LIN {X 0,Y 145.986,Z 279.775,A -85,B 0,C 180,E1 -25805.523,E2 -25805.523} C_VEL
LIN {X 0,Y 143.96,Z 293.571,A -85,B 0,C 180,E1 -25806.6,E2 -25806.6} C_VEL
LIN {X 0,Y 141.469,Z 306.049,A -85,B 0,C 180,E1 -25808.124,E2 -25808.124} C_VEL
LIN {X 0,Y 138.489,Z 317.193,A -85,B 0,C 180,E1 -25809.967,E2 -25809.967} C_VEL
LIN {X 0,Y 134.632,Z 328.9,A -85,B 0,C 180,E1 -25812.532,E2 -25812.532} C_VEL
LIN {X 0,Y 130.68,Z 339.104,A -85,B 0,C 180,E1 -25815.465,E2 -25815.465} C_VEL
LIN {X 0,Y 126.897,Z 348.015,A -85,B 0,C 180,E1 -25818.822,E2 -25818.822} C_VEL
LIN {X 0,Y 122.512,Z 357.337,A -85,B 0,C 180,E1 -25823.411,E2 -25823.411} C_VEL
LIN {X 0,Y 118.844,Z 364.909,A -85,B 0,C 180,E1 -25828.379,E2 -25828.379} C_VEL
LIN {X 0,Y 115.988,Z 370.741,A -85,B 0,C 180,E1 -25833.473,E2 -25833.473} C_VEL
LIN {X 0,Y 113.868,Z 375.53,A -85,B 0,C 180,E1 -25839.077,E2 -25839.077} C_VEL
LIN {X 0,Y 112.513,Z 378.89,A -85,B 0,C 180,E1 -25844.468,E2 -25844.468} C_VEL
LIN {X 0,Y 111.937,Z 381.142,A -85,B 0,C 180,E1 -25849.658,E2 -25849.658} C_VEL
LIN {X 0,Y 112.099,Z 382.715,A -85,B 0,C 180,E1 -25856.031,E2 -25856.031} C_VEL
LIN {X 0,Y 112.714,Z 383.083,A -85,B 0,C 180,E1 -25859.921,E2 -25859.921} C_VEL
LIN {X 0,Y 113.719,Z 382.989,A -85,B 0,C 180,E1 -25863.794,E2 -25863.794} C_VEL
LIN {X 0,Y 115.187,Z 382.397,A -85,B 0,C 180,E1 -25867.599,E2 -25867.599} C_VEL
LIN {X 0,Y 117.047,Z 381.361,A -85,B 0,C 180,E1 -25871.336,E2 -25871.336} C_VEL
LIN {X 0,Y 120.63,Z 378.856,A -85,B 0,C 180,E1 -25876.738,E2 -25876.738} C_VEL
LIN {X 0,Y 125.188,Z 375.1,A -85,B 0,C 180,E1 -25881.867,E2 -25881.867} C_VEL
LIN {X 0,Y 130.446,Z 370.145,A -85,B 0,C 180,E1 -25886.5,E2 -25886.5} C_VEL
LIN {X 0,Y 136.756,Z 363.485,A -85,B 0,C 180,E1 -25890.884,E2 -25890.884} C_VEL
LIN {X 0,Y 142.45,Z 356.634,A -85,B 0,C 180,E1 -25894.209,E2 -25894.209} C_VEL
LIN {X 0,Y 148.493,Z 348.43,A -85,B 0,C 180,E1 -25897.193,E2 -25897.193} C_VEL
LIN {X 0,Y 154.45,Z 338.924,A -85,B 0,C 180,E1 -25899.801,E2 -25899.801} C_VEL
LIN {X 0,Y 160.006,Z 328.535,A -85,B 0,C 180,E1 -25901.931,E2 -25901.931} C_VEL
LIN {X 0,Y 164.808,Z 317.654,A -85,B 0,C 180,E1 -25903.633,E2 -25903.633} C_VEL
LIN {X 0,Y 168.622,Z 306.885,A -85,B 0,C 180,E1 -25904.913,E2 -25904.913} C_VEL
LIN {X 0,Y 172.048,Z 293.907,A -85,B 0,C 180,E1 -25906.049,E2 -25906.049} C_VEL
LIN {X 0,Y 174.424,Z 281.013,A -85,B 0,C 180,E1 -25906.778,E2 -25906.778} C_VEL
LIN {X 0,Y 176.77,Z 258.578,A -85,B 0,C 180,E1 -25907.541,E2 -25907.541} C_VEL
LIN {X 0,Y 173.643,Z 251.901,A -85,B 0,C 180,E1 -25910.486,E2 -25910.486} C_VEL
LIN {X 0,Y 171.117,Z 247.12,A -85,B 0,C 180,E1 -25913.202,E2 -25913.202} C_VEL
LIN {X 0,Y 169.506,Z 244.096,A -85,B 0,C 180,E1 -25915.245,E2 -25915.245} C_VEL
LIN {X 0,Y 168.036,Z 241.322,A -85,B 0,C 180,E1 -25917.404,E2 -25917.404} C_VEL
LIN {X 0,Y 165.952,Z 237.408,A -85,B 0,C 180,E1 -25921.359,E2 -25921.359} C_VEL
LIN {X 0,Y 164.008,Z 233.239,A -85,B 0,C 180,E1 -25929.872,E2 -25929.872} C_VEL
LIN {X 0,Y 163.962,Z 233.673,A -85,B 0,C 180,E1 -25931.717,E2 -25931.717} C_VEL
LIN {X 0,Y 165.845,Z 237.96,A -85,B 0,C 180,E1 -25940.094,E2 -25940.094} C_VEL
LIN {X 0,Y 166.766,Z 239.887,A -85,B 0,C 180,E1 -25942.101,E2 -25942.101} C_VEL
LIN {X 0,Y 168.245,Z 242.318,A -85,B 0,C 180,E1 -25944.531,E2 -25944.531} C_VEL
LIN {X 0,Y 170.324,Z 247.29,A -85,B 0,C 180,E1 -25947.577,E2 -25947.577} C_VEL
LIN {X 0,Y 172.572,Z 252.652,A -85,B 0,C 180,E1 -25950.247,E2 -25950.247} C_VEL
LIN {X 0,Y 175.387,Z 260.766,A -85,B 0,C 180,E1 -25953.254,E2 -25953.254} C_VEL
LIN {X 0,Y 176.349,Z 263.654,A -85,B 0,C 180,E1 -25954.176,E2 -25954.176} C_VEL
LIN {X 0,Y 173.818,Z 287.836,A -85,B 0,C 180,E1 -25955.046,E2 -25955.046} C_VEL
LIN {X 0,Y 171.228,Z 301.026,A -85,B 0,C 180,E1 -25955.774,E2 -25955.774} C_VEL
LIN {X 0,Y 167.566,Z 313.569,A -85,B 0,C 180,E1 -25956.757,E2 -25956.757} C_VEL
LIN {X 0,Y 162.982,Z 325.554,A -85,B 0,C 180,E1 -25958.098,E2 -25958.098} C_VEL
LIN {X 0,Y 157.717,Z 336.638,A -85,B 0,C 180,E1 -25959.766,E2 -25959.766} C_VEL
LIN {X 0,Y 152.225,Z 346.648,A -85,B 0,C 180,E1 -25961.887,E2 -25961.887} C_VEL
LIN {X 0,Y 145.678,Z 356.545,A -85,B 0,C 180,E1 -25964.636,E2 -25964.636} C_VEL
LIN {X 0,Y 138.987,Z 365.314,A -85,B 0,C 180,E1 -25967.934,E2 -25967.934} C_VEL
LIN {X 0,Y 132.924,Z 372.398,A -85,B 0,C 180,E1 -25971.593,E2 -25971.593} C_VEL
LIN {X 0,Y 126.85,Z 378.898,A -85,B 0,C 180,E1 -25976.356,E2 -25976.356} C_VEL
LIN {X 0,Y 122.22,Z 383.244,A -85,B 0,C 180,E1 -25980.741,E2 -25980.741} C_VEL
LIN {X 0,Y 118.416,Z 386.557,A -85,B 0,C 180,E1 -25985.453,E2 -25985.453} C_VEL
LIN {X 0,Y 114.696,Z 389.513,A -85,B 0,C 180,E1 -25992.16,E2 -25992.16} C_VEL
LIN {X 0,Y 113.54,Z 390.406,A -85,B 0,C 180,E1 -25995.665,E2 -25995.665} C_VEL
LIN {X 0,Y 112.267,Z 390.977,A -85,B 0,C 180,E1 -26002.808,E2 -26002.808} C_VEL
LIN {X 0,Y 112.199,Z 390.696,A -85,B 0,C 180,E1 -26006.409,E2 -26006.409} C_VEL
LIN {X 0,Y 112.393,Z 390.029,A -85,B 0,C 180,E1 -26010.001,E2 -26010.001} C_VEL
LIN {X 0,Y 112.211,Z 388.885,A -85,B 0,C 180,E1 -26013.592,E2 -26013.592} C_VEL
LIN {X 0,Y 112.526,Z 386.385,A -85,B 0,C 180,E1 -26018.984,E2 -26018.984} C_VEL
LIN {X 0,Y 113.513,Z 382.837,A -85,B 0,C 180,E1 -26024.34,E2 -26024.34} C_VEL
LIN {X 0,Y 115.322,Z 378.149,A -85,B 0,C 180,E1 -26029.585,E2 -26029.585} C_VEL
LIN {X 0,Y 118.066,Z 372.192,A -85,B 0,C 180,E1 -26034.626,E2 -26034.626} C_VEL
LIN {X 0,Y 121.163,Z 365.534,A -85,B 0,C 180,E1 -26038.983,E2 -26038.983} C_VEL
LIN {X 0,Y 125.108,Z 357.123,A -85,B 0,C 180,E1 -26043.211,E2 -26043.211} C_VEL
LIN {X 0,Y 129.16,Z 347.899,A -85,B 0,C 180,E1 -26046.767,E2 -26046.767} C_VEL
LIN {X 0,Y 130.848,Z 343.784,A -85,B 0,C 180,E1 -26048.07,E2 -26048.07} C_VEL
LIN {X 0,Y 132.173,Z 339.134,A -85,B 0,C 180,E1 -26049.556,E2 -26049.556} C_VEL
LIN {X 0,Y 132.686,Z 331.21,A -85,B 0,C 180,E1 -26052.14,E2 -26052.14} C_VEL
LIN {X 0,Y 133.11,Z 322.867,A -85,B 0,C 180,E1 -26054.455,E2 -26054.455} C_VEL
LIN {X 0,Y 134.225,Z 317.564,A -85,B 0,C 180,E1 -26055.467,E2 -26055.467} C_VEL
LIN {X 0,Y 137.116,Z 306.394,A -85,B 0,C 180,E1 -26056.921,E2 -26056.921} C_VEL
LIN {X 0,Y 139.525,Z 293.458,A -85,B 0,C 180,E1 -26058.121,E2 -26058.121} C_VEL
LIN {X 0,Y 140.978,Z 280.384,A -85,B 0,C 180,E1 -26058.888,E2 -26058.888} C_VEL
LIN {X 0,Y 143.348,Z 248.743,A -85,B 0,C 180,E1 -26060.277,E2 -26060.277} C_VEL
LIN {X 0,Y 140.143,Z 238.589,A -85,B 0,C 180,E1 -26062.259,E2 -26062.259} C_VEL
LIN {X 0,Y 135.355,Z 226.534,A -85,B 0,C 180,E1 -26065.28,E2 -26065.28} C_VEL
LIN {X 0,Y 131.392,Z 217.778,A -85,B 0,C 180,E1 -26067.979,E2 -26067.979} C_VEL
LIN {X 0,Y 125.669,Z 208.745,A -85,B 0,C 180,E1 -26072.069,E2 -26072.069} C_VEL
LIN {X 0,Y 122.802,Z 204.727,A -85,B 0,C 180,E1 -26074.378,E2 -26074.378} C_VEL
LIN {X 0,Y 120.101,Z 200.884,A -85,B 0,C 180,E1 -26076.755,E2 -26076.755} C_VEL
LIN {X 0,Y 117.536,Z 197.763,A -85,B 0,C 180,E1 -26079.202,E2 -26079.202} C_VEL
LIN {X 0,Y 116.453,Z 196.028,A -85,B 0,C 180,E1 -26080.382,E2 -26080.382} C_VEL
LIN {X 0,Y 113.988,Z 193.648,A -85,B 0,C 180,E1 -26083.083,E2 -26083.083} C_VEL
LIN {X 0,Y 112.537,Z 190.796,A -85,B 0,C 180,E1 -26085.069,E2 -26085.069} C_VEL
LIN {X 0,Y 109.957,Z 188.848,A -85,B 0,C 180,E1 -26088.575,E2 -26088.575} C_VEL
LIN {X 0,Y 108.543,Z 186.343,A -85,B 0,C 180,E1 -26091.151,E2 -26091.151} C_VEL
LIN {X 0,Y 108.268,Z 184.955,A -85,B 0,C 180,E1 -26092.068,E2 -26092.068} C_VEL
LIN {X 0,Y 108.9,Z 184.896,A -85,B 0,C 180,E1 -26099.997,E2 -26099.997} C_VEL
LIN {X 0,Y 108.292,Z 184.978,A -85,B 0,C 180,E1 -26107.455,E2 -26107.455} C_VEL
LIN {X 0,Y 108.139,Z 184.981,A -85,B 0,C 180,E1 -26112.87,E2 -26112.87} C_VEL
LIN {X 0,Y 107.859,Z 185.022,A -85,B 0,C 180,E1 -26119.01,E2 -26119.01} C_VEL
LIN {X 0,Y 107.801,Z 185.034,A -85,B 0,C 180,E1 -26124.114,E2 -26124.114} C_VEL
LIN {X 0,Y 107.787,Z 185.047,A -85,B 0,C 180,E1 -26129.944,E2 -26129.944} C_VEL
LIN {X 0,Y 108.51,Z 187.423,A -85,B 0,C 180,E1 -26131.647,E2 -26131.647} C_VEL
LIN {X 0,Y 110.636,Z 189.968,A -85,B 0,C 180,E1 -26135.129,E2 -26135.129} C_VEL
LIN {X 0,Y 112.558,Z 191.06,A -85,B 0,C 180,E1 -26137.607,E2 -26137.607} C_VEL
LIN {X 0,Y 114.12,Z 193.989,A -85,B 0,C 180,E1 -26139.708,E2 -26139.708} C_VEL
LIN {X 0,Y 116.764,Z 196.565,A -85,B 0,C 180,E1 -26142.579,E2 -26142.579} C_VEL
LIN {X 0,Y 119.043,Z 200.028,A -85,B 0,C 180,E1 -26144.939,E2 -26144.939} C_VEL
LIN {X 0,Y 120.634,Z 201.729,A -85,B 0,C 180,E1 -26146.364,E2 -26146.364} C_VEL
LIN {X 0,Y 124.148,Z 206.696,A -85,B 0,C 180,E1 -26149.35,E2 -26149.35} C_VEL
LIN {X 0,Y 128.72,Z 213.396,A -85,B 0,C 180,E1 -26152.8,E2 -26152.8} C_VEL
LIN {X 0,Y 134.828,Z 223.62,A -85,B 0,C 180,E1 -26156.836,E2 -26156.836} C_VEL
LIN {X 0,Y 140.731,Z 234.972,A -85,B 0,C 180,E1 -26160.317,E2 -26160.317} C_VEL
LIN {X 0,Y 143.827,Z 241.661,A -85,B 0,C 180,E1 -26162.006,E2 -26162.006} C_VEL
LIN {X 0,Y 140.706,Z 279.337,A -85,B 0,C 180,E1 -26163.637,E2 -26163.637} C_VEL
LIN {X 0,Y 138.696,Z 292.716,A -85,B 0,C 180,E1 -26164.663,E2 -26164.663} C_VEL
LIN {X 0,Y 136.078,Z 305.504,A -85,B 0,C 180,E1 -26166.203,E2 -26166.203} C_VEL
LIN {X 0,Y 132.691,Z 317.65,A -85,B 0,C 180,E1 -26168.237,E2 -26168.237} C_VEL
LIN {X 0,Y 128.676,Z 329.311,A -85,B 0,C 180,E1 -26170.87,E2 -26170.87} C_VEL
LIN {X 0,Y 124.819,Z 338.762,A -85,B 0,C 180,E1 -26173.648,E2 -26173.648} C_VEL
LIN {X 0,Y 120.554,Z 348.369,A -85,B 0,C 180,E1 -26177.371,E2 -26177.371} C_VEL
LIN {X 0,Y 115.939,Z 357.673,A -85,B 0,C 180,E1 -26182.16,E2 -26182.16} C_VEL
LIN {X 0,Y 112.656,Z 364.034,A -85,B 0,C 180,E1 -26186.463,E2 -26186.463} C_VEL
LIN {X 0,Y 109.483,Z 370.163,A -85,B 0,C 180,E1 -26191.839,E2 -26191.839} C_VEL
LIN {X 0,Y 107.176,Z 375.01,A -85,B 0,C 180,E1 -26197.535,E2 -26197.535} C_VEL
LIN {X 0,Y 105.595,Z 378.69,A -85,B 0,C 180,E1 -26203.47,E2 -26203.47} C_VEL
LIN {X 0,Y 104.822,Z 381.467,A -85,B 0,C 180,E1 -26210.183,E2 -26210.183} C_VEL
LIN {X 0,Y 105.241,Z 383.128,A -85,B 0,C 180,E1 -26217.869,E2 -26217.869} C_VEL
LIN {X 0,Y 106.041,Z 383.377,A -85,B 0,C 180,E1 -26222.019,E2 -26222.019} C_VEL
LIN {X 0,Y 108.552,Z 382.675,A -85,B 0,C 180,E1 -26229.026,E2 -26229.026} C_VEL
LIN {X 0,Y 111.246,Z 381.268,A -85,B 0,C 180,E1 -26234.021,E2 -26234.021} C_VEL
LIN {X 0,Y 115.363,Z 378.544,A -85,B 0,C 180,E1 -26239.597,E2 -26239.597} C_VEL
LIN {X 0,Y 120.416,Z 374.603,A -85,B 0,C 180,E1 -26244.795,E2 -26244.795} C_VEL
LIN {X 0,Y 125.771,Z 369.863,A -85,B 0,C 180,E1 -26249.14,E2 -26249.14} C_VEL
LIN {X 0,Y 131.948,Z 363.75,A -85,B 0,C 180,E1 -26253.145,E2 -26253.145} C_VEL
LIN {X 0,Y 137.968,Z 356.91,A -85,B 0,C 180,E1 -26256.478,E2 -26256.478} C_VEL
LIN {X 0,Y 144.054,Z 349.03,A -85,B 0,C 180,E1 -26259.361,E2 -26259.361} C_VEL
LIN {X 0,Y 150.534,Z 339.207,A -85,B 0,C 180,E1 -26262.035,E2 -26262.035} C_VEL
LIN {X 0,Y 156.561,Z 328.354,A -85,B 0,C 180,E1 -26264.211,E2 -26264.211} C_VEL
LIN {X 0,Y 161.296,Z 317.944,A -85,B 0,C 180,E1 -26265.807,E2 -26265.807} C_VEL
LIN {X 0,Y 165.379,Z 306.809,A -85,B 0,C 180,E1 -26267.098,E2 -26267.098} C_VEL
LIN {X 0,Y 168.937,Z 293.767,A -85,B 0,C 180,E1 -26268.201,E2 -26268.201} C_VEL
LIN {X 0,Y 171.318,Z 281.228,A -85,B 0,C 180,E1 -26268.889,E2 -26268.889} C_VEL
LIN {X 0,Y 173.408,Z 262.063,A -85,B 0,C 180,E1 -26269.548,E2 -26269.548} C_VEL
LIN {X 0,Y 170.005,Z 254.678,A -85,B 0,C 180,E1 -26273.251,E2 -26273.251} C_VEL
LIN {X 0,Y 167.444,Z 249.727,A -85,B 0,C 180,E1 -26276.718,E2 -26276.718} C_VEL
LIN {X 0,Y 166.375,Z 247.659,A -85,B 0,C 180,E1 -26278.454,E2 -26278.454} C_VEL
LIN {X 0,Y 164.656,Z 244.108,A -85,B 0,C 180,E1 -26282.134,E2 -26282.134} C_VEL
LIN {X 0,Y 163.074,Z 240.291,A -85,B 0,C 180,E1 -26289.929,E2 -26289.929} C_VEL
LIN {X 0,Y 163.029,Z 241.202,A -85,B 0,C 180,E1 -26292.449,E2 -26292.449} C_VEL
LIN {X 0,Y 164.921,Z 245.281,A -85,B 0,C 180,E1 -26300.2,E2 -26300.2} C_VEL
LIN {X 0,Y 166.736,Z 248.974,A -85,B 0,C 180,E1 -26303.769,E2 -26303.769} C_VEL
LIN {X 0,Y 168.544,Z 253.593,A -85,B 0,C 180,E1 -26306.645,E2 -26306.645} C_VEL
LIN {X 0,Y 170.618,Z 259.175,A -85,B 0,C 180,E1 -26309.371,E2 -26309.371} C_VEL
LIN {X 0,Y 173.009,Z 266.682,A -85,B 0,C 180,E1 -26312.165,E2 -26312.165} C_VEL
LIN {X 0,Y 170.736,Z 287.3,A -85,B 0,C 180,E1 -26312.901,E2 -26312.901} C_VEL
LIN {X 0,Y 167.957,Z 301.038,A -85,B 0,C 180,E1 -26313.648,E2 -26313.648} C_VEL
LIN {X 0,Y 164.141,Z 313.583,A -85,B 0,C 180,E1 -26314.604,E2 -26314.604} C_VEL
LIN {X 0,Y 159.437,Z 325.465,A -85,B 0,C 180,E1 -26315.907,E2 -26315.907} C_VEL
LIN {X 0,Y 153.989,Z 336.517,A -85,B 0,C 180,E1 -26317.535,E2 -26317.535} C_VEL
LIN {X 0,Y 148.251,Z 346.498,A -85,B 0,C 180,E1 -26319.615,E2 -26319.615} C_VEL
LIN {X 0,Y 141.99,Z 355.572,A -85,B 0,C 180,E1 -26322.06,E2 -26322.06} C_VEL
LIN {X 0,Y 134.953,Z 364.447,A -85,B 0,C 180,E1 -26325.329,E2 -26325.329} C_VEL
LIN {X 0,Y 128.454,Z 371.634,A -85,B 0,C 180,E1 -26328.964,E2 -26328.964} C_VEL
LIN {X 0,Y 122.72,Z 377.421,A -85,B 0,C 180,E1 -26333.038,E2 -26333.038} C_VEL
LIN {X 0,Y 117.679,Z 382.027,A -85,B 0,C 180,E1 -26337.487,E2 -26337.487} C_VEL
LIN {X 0,Y 113.258,Z 385.576,A -85,B 0,C 180,E1 -26342.265,E2 -26342.265} C_VEL
LIN {X 0,Y 109.708,Z 388.155,A -85,B 0,C 180,E1 -26347.396,E2 -26347.396} C_VEL
LIN {X 0,Y 107.918,Z 389.392,A -85,B 0,C 180,E1 -26350.998,E2 -26350.998} C_VEL
LIN {X 0,Y 105.755,Z 390.64,A -85,B 0,C 180,E1 -26358.501,E2 -26358.501} C_VEL
LIN {X 0,Y 105.107,Z 390.377,A -85,B 0,C 180,E1 -26366.167,E2 -26366.167} C_VEL
LIN {X 0,Y 105.307,Z 389.652,A -85,B 0,C 180,E1 -26370.001,E2 -26370.001} C_VEL
LIN {X 0,Y 105.119,Z 388.453,A -85,B 0,C 180,E1 -26373.834,E2 -26373.834} C_VEL
LIN {X 0,Y 105.509,Z 385.873,A -85,B 0,C 180,E1 -26379.587,E2 -26379.587} C_VEL
LIN {X 0,Y 106.594,Z 382.236,A -85,B 0,C 180,E1 -26385.292,E2 -26385.292} C_VEL
LIN {X 0,Y 108.642,Z 377.46,A -85,B 0,C 180,E1 -26390.843,E2 -26390.843} C_VEL
LIN {X 0,Y 111.585,Z 371.396,A -85,B 0,C 180,E1 -26396.161,E2 -26396.161} C_VEL
LIN {X 0,Y 114.585,Z 365.353,A -85,B 0,C 180,E1 -26400.279,E2 -26400.279} C_VEL
LIN {X 0,Y 119.175,Z 356.083,A -85,B 0,C 180,E1 -26405.099,E2 -26405.099} C_VEL
LIN {X 0,Y 123.518,Z 346.651,A -85,B 0,C 180,E1 -26408.748,E2 -26408.748} C_VEL
LIN {X 0,Y 127.913,Z 336.182,A -85,B 0,C 180,E1 -26411.775,E2 -26411.775} C_VEL
LIN {X 0,Y 132.068,Z 324.552,A -85,B 0,C 180,E1 -26414.304,E2 -26414.304} C_VEL
LIN {X 0,Y 134.225,Z 317.564,A -85,B 0,C 180,E1 -26415.467,E2 -26415.467} C_VEL
LIN {X 0,Y 134.75,Z 313.661,A -85,B 0,C 180,E1 -26416.23,E2 -26416.23} C_VEL
LIN {X 0,Y 133.048,Z 302.423,A -85,B 0,C 180,E1 -26419.114,E2 -26419.114} C_VEL
LIN {X 0,Y 133.322,Z 298.652,A -85,B 0,C 180,E1 -26419.647,E2 -26419.647} C_VEL
LIN {X 0,Y 135.151,Z 286.464,A -85,B 0,C 180,E1 -26420.558,E2 -26420.558} C_VEL
LIN {X 0,Y 138.1,Z 250.25,A -85,B 0,C 180,E1 -26422.206,E2 -26422.206} C_VEL
LIN {X 0,Y 134.343,Z 238.888,A -85,B 0,C 180,E1 -26424.731,E2 -26424.731} C_VEL
LIN {X 0,Y 129.273,Z 226.193,A -85,B 0,C 180,E1 -26428.331,E2 -26428.331} C_VEL
LIN {X 0,Y 126.996,Z 221.599,A -85,B 0,C 180,E1 -26430.011,E2 -26430.011} C_VEL
LIN {X 0,Y 121.975,Z 213.498,A -85,B 0,C 180,E1 -26433.988,E2 -26433.988} C_VEL
LIN {X 0,Y 117.493,Z 206.959,A -85,B 0,C 180,E1 -26438.067,E2 -26438.067} C_VEL
LIN {X 0,Y 114.879,Z 203.515,A -85,B 0,C 180,E1 -26440.799,E2 -26440.799} C_VEL
LIN {X 0,Y 114.009,Z 202.24,A -85,B 0,C 180,E1 -26441.813,E2 -26441.813} C_VEL
LIN {X 0,Y 111.546,Z 199.443,A -85,B 0,C 180,E1 -26444.787,E2 -26444.787} C_VEL
LIN {X 0,Y 110.439,Z 197.355,A -85,B 0,C 180,E1 -26446.417,E2 -26446.417} C_VEL
LIN {X 0,Y 107.981,Z 195.031,A -85,B 0,C 180,E1 -26450.16,E2 -26450.16} C_VEL
LIN {X 0,Y 106.553,Z 192.054,A -85,B 0,C 180,E1 -26453.132,E2 -26453.132} C_VEL
LIN {X 0,Y 103.837,Z 189.952,A -85,B 0,C 180,E1 -26459.754,E2 -26459.754} C_VEL
LIN {X 0,Y 102.207,Z 188.654,A -85,B 0,C 180,E1 -26467.901,E2 -26467.901} C_VEL
LIN {X 0,Y 102.101,Z 188.838,A -85,B 0,C 180,E1 -26473.645,E2 -26473.645} C_VEL
LIN {X 0,Y 106.16,Z 192.173,A -85,B 0,C 180,E1 -26488.814,E2 -26488.814} C_VEL
LIN {X 0,Y 107.533,Z 195.102,A -85,B 0,C 180,E1 -26491.774,E2 -26491.774} C_VEL
LIN {X 0,Y 109.991,Z 197.293,A -85,B 0,C 180,E1 -26495.632,E2 -26495.632} C_VEL
LIN {X 0,Y 110.598,Z 197.854,A -85,B 0,C 180,E1 -26496.474,E2 -26496.474} C_VEL
LIN {X 0,Y 112.763,Z 201.229,A -85,B 0,C 180,E1 -26499.412,E2 -26499.412} C_VEL
LIN {X 0,Y 114.487,Z 202.991,A -85,B 0,C 180,E1 -26501.362,E2 -26501.362} C_VEL
LIN {X 0,Y 117.016,Z 206.654,A -85,B 0,C 180,E1 -26504.112,E2 -26504.112} C_VEL
LIN {X 0,Y 118.159,Z 208.076,A -85,B 0,C 180,E1 -26505.219,E2 -26505.219} C_VEL
LIN {X 0,Y 121.285,Z 212.635,A -85,B 0,C 180,E1 -26508.061,E2 -26508.061} C_VEL
LIN {X 0,Y 125.47,Z 218.96,A -85,B 0,C 180,E1 -26511.442,E2 -26511.442} C_VEL
LIN {X 0,Y 131.311,Z 229.167,A -85,B 0,C 180,E1 -26515.596,E2 -26515.596} C_VEL
LIN {X 0,Y 136.18,Z 238.872,A -85,B 0,C 180,E1 -26518.7,E2 -26518.7} C_VEL
LIN {X 0,Y 138.506,Z 243.986,A -85,B 0,C 180,E1 -26520.091,E2 -26520.091} C_VEL
LIN {X 0,Y 135.339,Z 280.315,A -85,B 0,C 180,E1 -26521.706,E2 -26521.706} C_VEL
LIN {X 0,Y 133.168,Z 294.058,A -85,B 0,C 180,E1 -26522.816,E2 -26522.816} C_VEL
LIN {X 0,Y 130.288,Z 306.924,A -85,B 0,C 180,E1 -26524.434,E2 -26524.434} C_VEL
LIN {X 0,Y 126.493,Z 319.61,A -85,B 0,C 180,E1 -26526.679,E2 -26526.679} C_VEL
LIN {X 0,Y 122.312,Z 330.947,A -85,B 0,C 180,E1 -26529.393,E2 -26529.393} C_VEL
LIN {X 0,Y 117.7,Z 341.534,A -85,B 0,C 180,E1 -26532.809,E2 -26532.809} C_VEL
LIN {X 0,Y 113.405,Z 350.362,A -85,B 0,C 180,E1 -26536.561,E2 -26536.561} C_VEL
LIN {X 0,Y 109.416,Z 357.967,A -85,B 0,C 180,E1 -26540.759,E2 -26540.759} C_VEL
LIN {X 0,Y 105.338,Z 365.423,A -85,B 0,C 180,E1 -26546.174,E2 -26546.174} C_VEL
LIN {X 0,Y 102.086,Z 371.331,A -85,B 0,C 180,E1 -26551.972,E2 -26551.972} C_VEL
LIN {X 0,Y 99.561,Z 376.411,A -85,B 0,C 180,E1 -26558.811,E2 -26558.811} C_VEL
LIN {X 0,Y 98.674,Z 378.418,A -85,B 0,C 180,E1 -26562.337,E2 -26562.337} C_VEL
LIN {X 0,Y 97.969,Z 380.397,A -85,B 0,C 180,E1 -26566.675,E2 -26566.675} C_VEL
LIN {X 0,Y 97.692,Z 381.873,A -85,B 0,C 180,E1 -26571.081,E2 -26571.081} C_VEL
LIN {X 0,Y 97.844,Z 382.922,A -85,B 0,C 180,E1 -26575.529,E2 -26575.529} C_VEL
LIN {X 0,Y 98.765,Z 383.579,A -85,B 0,C 180,E1 -26581.368,E2 -26581.368} C_VEL
LIN {X 0,Y 101.132,Z 383.279,A -85,B 0,C 180,E1 -26588.714,E2 -26588.714} C_VEL
LIN {X 0,Y 103.189,Z 382.459,A -85,B 0,C 180,E1 -26592.927,E2 -26592.927} C_VEL
LIN {X 0,Y 107.3,Z 380.24,A -85,B 0,C 180,E1 -26599.086,E2 -26599.086} C_VEL
LIN {X 0,Y 112.186,Z 376.997,A -85,B 0,C 180,E1 -26604.527,E2 -26604.527} C_VEL
LIN {X 0,Y 118.12,Z 372.407,A -85,B 0,C 180,E1 -26609.624,E2 -26609.624} C_VEL
LIN {X 0,Y 124.911,Z 366.402,A -85,B 0,C 180,E1 -26614.187,E2 -26614.187} C_VEL
LIN {X 0,Y 132.107,Z 358.967,A -85,B 0,C 180,E1 -26618.14,E2 -26618.14} C_VEL
LIN {X 0,Y 139.091,Z 350.599,A -85,B 0,C 180,E1 -26621.333,E2 -26621.333} C_VEL
LIN {X 0,Y 146.136,Z 340.69,A -85,B 0,C 180,E1 -26624.12,E2 -26624.12} C_VEL
LIN {X 0,Y 152.654,Z 329.59,A -85,B 0,C 180,E1 -26626.369,E2 -26626.369} C_VEL
LIN {X 0,Y 158.03,Z 318.383,A -85,B 0,C 180,E1 -26628.067,E2 -26628.067} C_VEL
LIN {X 0,Y 162.263,Z 307.347,A -85,B 0,C 180,E1 -26629.311,E2 -26629.311} C_VEL
LIN {X 0,Y 165.934,Z 294.444,A -85,B 0,C 180,E1 -26630.383,E2 -26630.383} C_VEL
LIN {X 0,Y 168.464,Z 281.635,A -85,B 0,C 180,E1 -26631.073,E2 -26631.073} C_VEL
LIN {X 0,Y 170.269,Z 265.817,A -85,B 0,C 180,E1 -26631.627,E2 -26631.627} C_VEL
LIN {X 0,Y 167.851,Z 260.355,A -85,B 0,C 180,E1 -26634.614,E2 -26634.614} C_VEL
LIN {X 0,Y 165.304,Z 254.823,A -85,B 0,C 180,E1 -26638.591,E2 -26638.591} C_VEL
LIN {X 0,Y 163.471,Z 250.965,A -85,B 0,C 180,E1 -26642.7,E2 -26642.7} C_VEL
LIN {X 0,Y 162.142,Z 247.336,A -85,B 0,C 180,E1 -26649.986,E2 -26649.986} C_VEL
LIN {X 0,Y 162.174,Z 249.055,A -85,B 0,C 180,E1 -26653.808,E2 -26653.808} C_VEL
LIN {X 0,Y 163.712,Z 252.146,A -85,B 0,C 180,E1 -26659.638,E2 -26659.638} C_VEL
LIN {X 0,Y 165.203,Z 255.442,A -85,B 0,C 180,E1 -26662.885,E2 -26662.885} C_VEL
LIN {X 0,Y 166.911,Z 260.166,A -85,B 0,C 180,E1 -26665.843,E2 -26665.843} C_VEL
LIN {X 0,Y 169.071,Z 266.801,A -85,B 0,C 180,E1 -26668.952,E2 -26668.952} C_VEL
LIN {X 0,Y 169.939,Z 269.913,A -85,B 0,C 180,E1 -26670.091,E2 -26670.091} C_VEL
LIN {X 0,Y 167.742,Z 288.204,A -85,B 0,C 180,E1 -26670.739,E2 -26670.739} C_VEL
LIN {X 0,Y 165.238,Z 300.051,A -85,B 0,C 180,E1 -26671.362,E2 -26671.362} C_VEL
LIN {X 0,Y 161.798,Z 311.475,A -85,B 0,C 180,E1 -26672.176,E2 -26672.176} C_VEL
LIN {X 0,Y 157.555,Z 322.353,A -85,B 0,C 180,E1 -26673.241,E2 -26673.241} C_VEL
LIN {X 0,Y 151.898,Z 333.904,A -85,B 0,C 180,E1 -26674.79,E2 -26674.79} C_VEL
LIN {X 0,Y 145.798,Z 344.307,A -85,B 0,C 180,E1 -26676.738,E2 -26676.738} C_VEL
LIN {X 0,Y 138.639,Z 354.594,A -85,B 0,C 180,E1 -26679.371,E2 -26679.371} C_VEL
LIN {X 0,Y 131.18,Z 363.593,A -85,B 0,C 180,E1 -26682.553,E2 -26682.553} C_VEL
LIN {X 0,Y 124.291,Z 370.88,A -85,B 0,C 180,E1 -26686.159,E2 -26686.159} C_VEL
LIN {X 0,Y 117.111,Z 377.623,A -85,B 0,C 180,E1 -26690.942,E2 -26690.942} C_VEL
LIN {X 0,Y 111.74,Z 382.122,A -85,B 0,C 180,E1 -26695.525,E2 -26695.525} C_VEL
LIN {X 0,Y 108.44,Z 384.518,A -85,B 0,C 180,E1 -26698.77,E2 -26698.77} C_VEL
LIN {X 0,Y 103.182,Z 388.08,A -85,B 0,C 180,E1 -26705.879,E2 -26705.879} C_VEL
LIN {X 0,Y 101.194,Z 389.242,A -85,B 0,C 180,E1 -26709.681,E2 -26709.681} C_VEL
LIN {X 0,Y 98.772,Z 390.399,A -85,B 0,C 180,E1 -26717.676,E2 -26717.676} C_VEL
LIN {X 0,Y 98.017,Z 390.045,A -85,B 0,C 180,E1 -26725.889,E2 -26725.889} C_VEL
LIN {X 0,Y 98.207,Z 389.247,A -85,B 0,C 180,E1 -26730.001,E2 -26730.001} C_VEL
LIN {X 0,Y 98.029,Z 388.005,A -85,B 0,C 180,E1 -26734.112,E2 -26734.112} C_VEL
LIN {X 0,Y 98.492,Z 385.337,A -85,B 0,C 180,E1 -26740.277,E2 -26740.277} C_VEL
LIN {X 0,Y 99.723,Z 381.607,A -85,B 0,C 180,E1 -26746.375,E2 -26746.375} C_VEL
LIN {X 0,Y 101.997,Z 376.733,A -85,B 0,C 180,E1 -26752.271,E2 -26752.271} C_VEL
LIN {X 0,Y 105.211,Z 370.558,A -85,B 0,C 180,E1 -26757.879,E2 -26757.879} C_VEL
LIN {X 0,Y 107.853,Z 365.606,A -85,B 0,C 180,E1 -26761.421,E2 -26761.421} C_VEL
LIN {X 0,Y 112.553,Z 356.632,A -85,B 0,C 180,E1 -26766.385,E2 -26766.385} C_VEL
LIN {X 0,Y 117.057,Z 347.413,A -85,B 0,C 180,E1 -26770.198,E2 -26770.198} C_VEL
LIN {X 0,Y 121.603,Z 337.187,A -85,B 0,C 180,E1 -26773.34,E2 -26773.34} C_VEL
LIN {X 0,Y 125.943,Z 325.848,A -85,B 0,C 180,E1 -26775.929,E2 -26775.929} C_VEL
LIN {X 0,Y 129.712,Z 314.142,A -85,B 0,C 180,E1 -26777.87,E2 -26777.87} C_VEL
LIN {X 0,Y 132.746,Z 301.431,A -85,B 0,C 180,E1 -26779.396,E2 -26779.396} C_VEL
LIN {X 0,Y 133.322,Z 298.652,A -85,B 0,C 180,E1 -26779.647,E2 -26779.647} C_VEL
LIN {X 0,Y 133.843,Z 294.862,A -85,B 0,C 180,E1 -26780.04,E2 -26780.04} C_VEL
LIN {X 0,Y 133.687,Z 289.229,A -85,B 0,C 180,E1 -26780.831,E2 -26780.831} C_VEL
LIN {X 0,Y 131.637,Z 274.299,A -85,B 0,C 180,E1 -26783.068,E2 -26783.068} C_VEL
LIN {X 0,Y 131.714,Z 268.46,A -85,B 0,C 180,E1 -26783.499,E2 -26783.499} C_VEL
LIN {X 0,Y 133.024,Z 252.286,A -85,B 0,C 180,E1 -26784.233,E2 -26784.233} C_VEL
LIN {X 0,Y 129.62,Z 241.704,A -85,B 0,C 180,E1 -26786.773,E2 -26786.773} C_VEL
LIN {X 0,Y 124.752,Z 229.224,A -85,B 0,C 180,E1 -26790.579,E2 -26790.579} C_VEL
LIN {X 0,Y 121.72,Z 223.626,A -85,B 0,C 180,E1 -26793.063,E2 -26793.063} C_VEL
LIN {X 0,Y 117.327,Z 216.614,A -85,B 0,C 180,E1 -26797.011,E2 -26797.011} C_VEL
LIN {X 0,Y 114.586,Z 212.646,A -85,B 0,C 180,E1 -26799.815,E2 -26799.815} C_VEL
LIN {X 0,Y 111.739,Z 208.536,A -85,B 0,C 180,E1 -26803.163,E2 -26803.163} C_VEL
LIN {X 0,Y 109.249,Z 205.319,A -85,B 0,C 180,E1 -26806.481,E2 -26806.481} C_VEL
LIN {X 0,Y 108.548,Z 203.91,A -85,B 0,C 180,E1 -26807.623,E2 -26807.623} C_VEL
LIN {X 0,Y 106.113,Z 201.204,A -85,B 0,C 180,E1 -26811.756,E2 -26811.756} C_VEL
LIN {X 0,Y 104.865,Z 198.646,A -85,B 0,C 180,E1 -26814.577,E2 -26814.577} C_VEL
LIN {X 0,Y 102.813,Z 197.01,A -85,B 0,C 180,E1 -26819.997,E2 -26819.997} C_VEL
LIN {X 0,Y 101.272,Z 195.695,A -85,B 0,C 180,E1 -26827.975,E2 -26827.975} C_VEL
LIN {X 0,Y 101.169,Z 195.865,A -85,B 0,C 180,E1 -26833.45,E2 -26833.45} C_VEL
LIN {X 0,Y 104.664,Z 199.066,A -85,B 0,C 180,E1 -26847.761,E2 -26847.761} C_VEL
LIN {X 0,Y 106.33,Z 202.248,A -85,B 0,C 180,E1 -26851.451,E2 -26851.451} C_VEL
LIN {X 0,Y 108.698,Z 204.472,A -85,B 0,C 180,E1 -26855.286,E2 -26855.286} C_VEL
LIN {X 0,Y 111.184,Z 208.148,A -85,B 0,C 180,E1 -26858.819,E2 -26858.819} C_VEL
LIN {X 0,Y 112.421,Z 209.668,A -85,B 0,C 180,E1 -26860.321,E2 -26860.321} C_VEL
LIN {X 0,Y 115.046,Z 213.266,A -85,B 0,C 180,E1 -26863.283,E2 -26863.283} C_VEL
LIN {X 0,Y 118.616,Z 218.763,A -85,B 0,C 180,E1 -26866.842,E2 -26866.842} C_VEL
LIN {X 0,Y 122.21,Z 224.431,A -85,B 0,C 180,E1 -26869.951,E2 -26869.951} C_VEL
LIN {X 0,Y 127.262,Z 233.569,A -85,B 0,C 180,E1 -26873.877,E2 -26873.877} C_VEL
LIN {X 0,Y 132.714,Z 244.812,A -85,B 0,C 180,E1 -26877.608,E2 -26877.608} C_VEL
LIN {X 0,Y 133.419,Z 246.506,A -85,B 0,C 180,E1 -26878.076,E2 -26878.076} C_VEL
LIN {X 0,Y 130.266,Z 280.463,A -85,B 0,C 180,E1 -26879.572,E2 -26879.572} C_VEL
LIN {X 0,Y 127.96,Z 294.466,A -85,B 0,C 180,E1 -26880.714,E2 -26880.714} C_VEL
LIN {X 0,Y 124.941,Z 307.283,A -85,B 0,C 180,E1 -26882.349,E2 -26882.349} C_VEL
LIN {X 0,Y 120.973,Z 319.944,A -85,B 0,C 180,E1 -26884.63,E2 -26884.63} C_VEL
LIN {X 0,Y 116.569,Z 331.271,A -85,B 0,C 180,E1 -26887.396,E2 -26887.396} C_VEL
LIN {X 0,Y 111.906,Z 341.455,A -85,B 0,C 180,E1 -26890.755,E2 -26890.755} C_VEL
LIN {X 0,Y 107.184,Z 350.665,A -85,B 0,C 180,E1 -26894.794,E2 -26894.794} C_VEL
LIN {X 0,Y 102.957,Z 358.263,A -85,B 0,C 180,E1 -26899.179,E2 -26899.179} C_VEL
LIN {X 0,Y 98.826,Z 365.371,A -85,B 0,C 180,E1 -26904.586,E2 -26904.586} C_VEL
LIN {X 0,Y 95.669,Z 370.739,A -85,B 0,C 180,E1 -26909.999,E2 -26909.999} C_VEL
LIN {X 0,Y 93.086,Z 375.544,A -85,B 0,C 180,E1 -26916.454,E2 -26916.454} C_VEL
LIN {X 0,Y 91.336,Z 379.247,A -85,B 0,C 180,E1 -26923.346,E2 -26923.346} C_VEL
LIN {X 0,Y 90.584,Z 382.092,A -85,B 0,C 180,E1 -26931.416,E2 -26931.416} C_VEL
LIN {X 0,Y 90.946,Z 383.385,A -85,B 0,C 180,E1 -26937.623,E2 -26937.623} C_VEL
LIN {X 0,Y 91.912,Z 383.849,A -85,B 0,C 180,E1 -26942.749,E2 -26942.749} C_VEL
LIN {X 0,Y 93.203,Z 383.85,A -85,B 0,C 180,E1 -26947.102,E2 -26947.102} C_VEL
LIN {X 0,Y 95.696,Z 383.189,A -85,B 0,C 180,E1 -26952.748,E2 -26952.748} C_VEL
LIN {X 0,Y 100.528,Z 381.03,A -85,B 0,C 180,E1 -26960.265,E2 -26960.265} C_VEL
LIN {X 0,Y 105.815,Z 377.926,A -85,B 0,C 180,E1 -26966.121,E2 -26966.121} C_VEL
LIN {X 0,Y 112.052,Z 373.543,A -85,B 0,C 180,E1 -26971.412,E2 -26971.412} C_VEL
LIN {X 0,Y 119.537,Z 367.442,A -85,B 0,C 180,E1 -26976.313,E2 -26976.313} C_VEL
LIN {X 0,Y 126.957,Z 360.408,A -85,B 0,C 180,E1 -26980.232,E2 -26980.232} C_VEL
LIN {X 0,Y 133.908,Z 352.714,A -85,B 0,C 180,E1 -26983.3,E2 -26983.3} C_VEL
LIN {X 0,Y 141.403,Z 342.902,A -85,B 0,C 180,E1 -26986.147,E2 -26986.147} C_VEL
LIN {X 0,Y 148.011,Z 332.592,A -85,B 0,C 180,E1 -26988.331,E2 -26988.331} C_VEL
LIN {X 0,Y 153.512,Z 322.158,A -85,B 0,C 180,E1 -26989.966,E2 -26989.966} C_VEL
LIN {X 0,Y 158.589,Z 310.004,A -85,B 0,C 180,E1 -26991.413,E2 -26991.413} C_VEL
LIN {X 0,Y 162.437,Z 298.005,A -85,B 0,C 180,E1 -26992.443,E2 -26992.443} C_VEL
LIN {X 0,Y 165.247,Z 285.747,A -85,B 0,C 180,E1 -26993.167,E2 -26993.167} C_VEL
LIN {X 0,Y 167.161,Z 272.274,A -85,B 0,C 180,E1 -26993.625,E2 -26993.625} C_VEL
LIN {X 0,Y 167.368,Z 269.776,A -85,B 0,C 180,E1 -26993.765,E2 -26993.765} C_VEL
LIN {X 0,Y 165.151,Z 264.366,A -85,B 0,C 180,E1 -26997.076,E2 -26997.076} C_VEL
LIN {X 0,Y 163.568,Z 260.888,A -85,B 0,C 180,E1 -27000.002,E2 -27000.002} C_VEL
LIN {X 0,Y 162.335,Z 257.843,A -85,B 0,C 180,E1 -27003.191,E2 -27003.191} C_VEL
LIN {X 0,Y 161.193,Z 254.503,A -85,B 0,C 180,E1 -27010.046,E2 -27010.046} C_VEL
LIN {X 0,Y 161.209,Z 256.138,A -85,B 0,C 180,E1 -27013.623,E2 -27013.623} C_VEL
LIN {X 0,Y 162.504,Z 258.915,A -85,B 0,C 180,E1 -27019.008,E2 -27019.008} C_VEL
LIN {X 0,Y 163.714,Z 261.93,A -85,B 0,C 180,E1 -27021.989,E2 -27021.989} C_VEL
LIN {X 0,Y 165.11,Z 266.183,A -85,B 0,C 180,E1 -27024.687,E2 -27024.687} C_VEL
LIN {X 0,Y 166.782,Z 271.981,A -85,B 0,C 180,E1 -27027.468,E2 -27027.468} C_VEL
LIN {X 0,Y 167.112,Z 273.27,A -85,B 0,C 180,E1 -27027.973,E2 -27027.973} C_VEL
LIN {X 0,Y 164.914,Z 289.546,A -85,B 0,C 180,E1 -27028.515,E2 -27028.515} C_VEL
LIN {X 0,Y 161.774,Z 302.82,A -85,B 0,C 180,E1 -27029.235,E2 -27029.235} C_VEL
LIN {X 0,Y 157.497,Z 315.37,A -85,B 0,C 180,E1 -27030.167,E2 -27030.167} C_VEL
LIN {X 0,Y 152.347,Z 327.082,A -85,B 0,C 180,E1 -27031.413,E2 -27031.413} C_VEL
LIN {X 0,Y 146.57,Z 337.63,A -85,B 0,C 180,E1 -27032.953,E2 -27032.953} C_VEL
LIN {X 0,Y 139.701,Z 348.227,A -85,B 0,C 180,E1 -27035.166,E2 -27035.166} C_VEL
LIN {X 0,Y 132.957,Z 356.912,A -85,B 0,C 180,E1 -27037.544,E2 -27037.544} C_VEL
LIN {X 0,Y 125.289,Z 365.422,A -85,B 0,C 180,E1 -27040.776,E2 -27040.776} C_VEL
LIN {X 0,Y 118.128,Z 372.273,A -85,B 0,C 180,E1 -27044.444,E2 -27044.444} C_VEL
LIN {X 0,Y 111.682,Z 377.811,A -85,B 0,C 180,E1 -27048.643,E2 -27048.643} C_VEL
LIN {X 0,Y 105.95,Z 382.207,A -85,B 0,C 180,E1 -27053.346,E2 -27053.346} C_VEL
LIN {X 0,Y 102.429,Z 384.555,A -85,B 0,C 180,E1 -27056.709,E2 -27056.709} C_VEL
LIN {X 0,Y 99.401,Z 386.487,A -85,B 0,C 180,E1 -27060.336,E2 -27060.336} C_VEL
LIN {X 0,Y 96.743,Z 388,A -85,B 0,C 180,E1 -27064.16,E2 -27064.16} C_VEL
LIN {X 0,Y 92.943,Z 389.811,A -85,B 0,C 180,E1 -27072.395,E2 -27072.395} C_VEL
LIN {X 0,Y 91.139,Z 390.131,A -85,B 0,C 180,E1 -27081.129,E2 -27081.129} C_VEL
LIN {X 0,Y 90.924,Z 389.685,A -85,B 0,C 180,E1 -27085.568,E2 -27085.568} C_VEL
LIN {X 0,Y 91.118,Z 388.842,A -85,B 0,C 180,E1 -27090.001,E2 -27090.001} C_VEL
LIN {X 0,Y 90.937,Z 387.557,A -85,B 0,C 180,E1 -27094.433,E2 -27094.433} C_VEL
LIN {X 0,Y 91.5,Z 384.801,A -85,B 0,C 180,E1 -27101.072,E2 -27101.072} C_VEL
LIN {X 0,Y 92.898,Z 380.976,A -85,B 0,C 180,E1 -27107.616,E2 -27107.616} C_VEL
LIN {X 0,Y 95.426,Z 376.001,A -85,B 0,C 180,E1 -27113.897,E2 -27113.897} C_VEL
LIN {X 0,Y 98.958,Z 369.717,A -85,B 0,C 180,E1 -27119.812,E2 -27119.812} C_VEL
LIN {X 0,Y 102.993,Z 362.474,A -85,B 0,C 180,E1 -27124.929,E2 -27124.929} C_VEL
LIN {X 0,Y 107.778,Z 353.758,A -85,B 0,C 180,E1 -27129.479,E2 -27129.479} C_VEL
LIN {X 0,Y 112.697,Z 343.907,A -85,B 0,C 180,E1 -27133.314,E2 -27133.314} C_VEL
LIN {X 0,Y 117.68,Z 332.979,A -85,B 0,C 180,E1 -27136.397,E2 -27136.397} C_VEL
LIN {X 0,Y 121.618,Z 322.21,A -85,B 0,C 180,E1 -27138.699,E2 -27138.699} C_VEL
LIN {X 0,Y 125.641,Z 309.392,A -85,B 0,C 180,E1 -27140.592,E2 -27140.592} C_VEL
LIN {X 0,Y 128.495,Z 296.753,A -85,B 0,C 180,E1 -27141.924,E2 -27141.924} C_VEL
LIN {X 0,Y 130.384,Z 283.274,A -85,B 0,C 180,E1 -27142.844,E2 -27142.844} C_VEL
LIN {X 0,Y 131.714,Z 268.46,A -85,B 0,C 180,E1 -27143.499,E2 -27143.499} C_VEL
LIN {X 0,Y 131.656,Z 264.622,A -85,B 0,C 180,E1 -27143.841,E2 -27143.841} C_VEL
LIN {X 0,Y 130.9,Z 261.019,A -85,B 0,C 180,E1 -27144.489,E2 -27144.489} C_VEL
LIN {X 0,Y 126.79,Z 249.802,A -85,B 0,C 180,E1 -27147.498,E2 -27147.498} C_VEL
LIN {X 0,Y 122.248,Z 236.886,A -85,B 0,C 180,E1 -27151.333,E2 -27151.333} C_VEL
LIN {X 0,Y 120.109,Z 231.891,A -85,B 0,C 180,E1 -27153.254,E2 -27153.254} C_VEL
LIN {X 0,Y 115.609,Z 224.068,A -85,B 0,C 180,E1 -27157.461,E2 -27157.461} C_VEL
LIN {X 0,Y 112.225,Z 218.798,A -85,B 0,C 180,E1 -27161.158,E2 -27161.158} C_VEL
LIN {X 0,Y 109.444,Z 214.699,A -85,B 0,C 180,E1 -27164.663,E2 -27164.663} C_VEL
LIN {X 0,Y 107.015,Z 211.107,A -85,B 0,C 180,E1 -27168.31,E2 -27168.31} C_VEL
LIN {X 0,Y 106.303,Z 210.107,A -85,B 0,C 180,E1 -27169.522,E2 -27169.522} C_VEL
LIN {X 0,Y 104.062,Z 206.95,A -85,B 0,C 180,E1 -27173.938,E2 -27173.938} C_VEL
LIN {X 0,Y 103.382,Z 205.465,A -85,B 0,C 180,E1 -27175.699,E2 -27175.699} C_VEL
LIN {X 0,Y 101.337,Z 203.637,A -85,B 0,C 180,E1 -27181.984,E2 -27181.984} C_VEL
LIN {X 0,Y 100.336,Z 202.744,A -85,B 0,C 180,E1 -27188.05,E2 -27188.05} C_VEL
LIN {X 0,Y 100.238,Z 202.976,A -85,B 0,C 180,E1 -27193.577,E2 -27193.577} C_VEL
LIN {X 0,Y 103.216,Z 205.86,A -85,B 0,C 180,E1 -27206.674,E2 -27206.674} C_VEL
LIN {X 0,Y 104.981,Z 209.168,A -85,B 0,C 180,E1 -27210.833,E2 -27210.833} C_VEL
LIN {X 0,Y 106.874,Z 211.066,A -85,B 0,C 180,E1 -27214.092,E2 -27214.092} C_VEL
LIN {X 0,Y 109.575,Z 214.986,A -85,B 0,C 180,E1 -27218.15,E2 -27218.15} C_VEL
LIN {X 0,Y 113.434,Z 220.758,A -85,B 0,C 180,E1 -27222.852,E2 -27222.852} C_VEL
LIN {X 0,Y 117.541,Z 227.305,A -85,B 0,C 180,E1 -27227.039,E2 -27227.039} C_VEL
LIN {X 0,Y 122.295,Z 235.915,A -85,B 0,C 180,E1 -27231.202,E2 -27231.202} C_VEL
LIN {X 0,Y 127.616,Z 247.082,A -85,B 0,C 180,E1 -27235.3,E2 -27235.3} C_VEL
LIN {X 0,Y 128.411,Z 248.87,A -85,B 0,C 180,E1 -27235.866,E2 -27235.866} C_VEL
LIN {X 0,Y 125.383,Z 280.457,A -85,B 0,C 180,E1 -27237.272,E2 -27237.272} C_VEL
LIN {X 0,Y 122.999,Z 294.422,A -85,B 0,C 180,E1 -27238.405,E2 -27238.405} C_VEL
LIN {X 0,Y 120.096,Z 306.506,A -85,B 0,C 180,E1 -27239.928,E2 -27239.928} C_VEL
LIN {X 0,Y 116.204,Z 318.591,A -85,B 0,C 180,E1 -27242.048,E2 -27242.048} C_VEL
LIN {X 0,Y 111.582,Z 330.216,A -85,B 0,C 180,E1 -27244.839,E2 -27244.839} C_VEL
LIN {X 0,Y 106.595,Z 340.702,A -85,B 0,C 180,E1 -27248.234,E2 -27248.234} C_VEL
LIN {X 0,Y 101.092,Z 350.919,A -85,B 0,C 180,E1 -27252.814,E2 -27252.814} C_VEL
LIN {X 0,Y 96.584,Z 358.521,A -85,B 0,C 180,E1 -27257.39,E2 -27257.39} C_VEL
LIN {X 0,Y 91.962,Z 365.98,A -85,B 0,C 180,E1 -27263.43,E2 -27263.43} C_VEL
LIN {X 0,Y 88.284,Z 371.869,A -85,B 0,C 180,E1 -27269.999,E2 -27269.999} C_VEL
LIN {X 0,Y 85.82,Z 376.214,A -85,B 0,C 180,E1 -27276.551,E2 -27276.551} C_VEL
LIN {X 0,Y 84.015,Z 379.989,A -85,B 0,C 180,E1 -27284.533,E2 -27284.533} C_VEL
LIN {X 0,Y 83.517,Z 382.405,A -85,B 0,C 180,E1 -27292.244,E2 -27292.244} C_VEL
LIN {X 0,Y 84.191,Z 383.793,A -85,B 0,C 180,E1 -27300.056,E2 -27300.056} C_VEL
LIN {X 0,Y 85.373,Z 384.157,A -85,B 0,C 180,E1 -27305.186,E2 -27305.186} C_VEL
LIN {X 0,Y 87.098,Z 384.048,A -85,B 0,C 180,E1 -27310.204,E2 -27310.204} C_VEL
LIN {X 0,Y 89.447,Z 383.452,A -85,B 0,C 180,E1 -27315.002,E2 -27315.002} C_VEL
LIN {X 0,Y 92.302,Z 382.411,A -85,B 0,C 180,E1 -27319.588,E2 -27319.588} C_VEL
LIN {X 0,Y 95.874,Z 380.755,A -85,B 0,C 180,E1 -27324.1,E2 -27324.1} C_VEL
LIN {X 0,Y 101.62,Z 377.547,A -85,B 0,C 180,E1 -27329.824,E2 -27329.824} C_VEL
LIN {X 0,Y 108.511,Z 372.979,A -85,B 0,C 180,E1 -27335.058,E2 -27335.058} C_VEL
LIN {X 0,Y 115.94,Z 367.224,A -85,B 0,C 180,E1 -27339.478,E2 -27339.478} C_VEL
LIN {X 0,Y 123.1,Z 360.74,A -85,B 0,C 180,E1 -27342.995,E2 -27342.995} C_VEL
LIN {X 0,Y 130.379,Z 353.067,A -85,B 0,C 180,E1 -27345.995,E2 -27345.995} C_VEL
LIN {X 0,Y 137.969,Z 343.57,A -85,B 0,C 180,E1 -27348.686,E2 -27348.686} C_VEL
LIN {X 0,Y 145.043,Z 333.031,A -85,B 0,C 180,E1 -27350.845,E2 -27350.845} C_VEL
LIN {X 0,Y 150.666,Z 322.806,A -85,B 0,C 180,E1 -27352.405,E2 -27352.405} C_VEL
LIN {X 0,Y 155.558,Z 311.74,A -85,B 0,C 180,E1 -27353.688,E2 -27353.688} C_VEL
LIN {X 0,Y 159.639,Z 299.808,A -85,B 0,C 180,E1 -27354.714,E2 -27354.714} C_VEL
LIN {X 0,Y 162.642,Z 287.748,A -85,B 0,C 180,E1 -27355.436,E2 -27355.436} C_VEL
LIN {X 0,Y 164.612,Z 275.558,A -85,B 0,C 180,E1 -27355.877,E2 -27355.877} C_VEL
LIN {X 0,Y 164.762,Z 273.865,A -85,B 0,C 180,E1 -27355.974,E2 -27355.974} C_VEL
LIN {X 0,Y 162.842,Z 269.013,A -85,B 0,C 180,E1 -27359.4,E2 -27359.4} C_VEL
LIN {X 0,Y 161.291,Z 264.856,A -85,B 0,C 180,E1 -27363.449,E2 -27363.449} C_VEL
LIN {X 0,Y 160.245,Z 261.667,A -85,B 0,C 180,E1 -27370.106,E2 -27370.106} C_VEL
LIN {X 0,Y 161.325,Z 265.762,A -85,B 0,C 180,E1 -27378.414,E2 -27378.414} C_VEL
LIN {X 0,Y 162.371,Z 268.644,A -85,B 0,C 180,E1 -27381.256,E2 -27381.256} C_VEL
LIN {X 0,Y 163.573,Z 272.807,A -85,B 0,C 180,E1 -27383.88,E2 -27383.88} C_VEL
LIN {X 0,Y 164.515,Z 276.584,A -85,B 0,C 180,E1 -27385.684,E2 -27385.684} C_VEL
LIN {X 0,Y 162.517,Z 290.181,A -85,B 0,C 180,E1 -27386.185,E2 -27386.185} C_VEL
LIN {X 0,Y 159.332,Z 302.953,A -85,B 0,C 180,E1 -27386.859,E2 -27386.859} C_VEL
LIN {X 0,Y 154.859,Z 315.598,A -85,B 0,C 180,E1 -27387.752,E2 -27387.752} C_VEL
LIN {X 0,Y 149.563,Z 327.157,A -85,B 0,C 180,E1 -27388.933,E2 -27388.933} C_VEL
LIN {X 0,Y 142.87,Z 338.771,A -85,B 0,C 180,E1 -27390.588,E2 -27390.588} C_VEL
LIN {X 0,Y 135.772,Z 349.133,A -85,B 0,C 180,E1 -27392.739,E2 -27392.739} C_VEL
LIN {X 0,Y 128.782,Z 357.616,A -85,B 0,C 180,E1 -27395.056,E2 -27395.056} C_VEL
LIN {X 0,Y 120.779,Z 365.903,A -85,B 0,C 180,E1 -27398.229,E2 -27398.229} C_VEL
LIN {X 0,Y 113.282,Z 372.62,A -85,B 0,C 180,E1 -27401.887,E2 -27401.887} C_VEL
LIN {X 0,Y 106.452,Z 378.027,A -85,B 0,C 180,E1 -27406.116,E2 -27406.116} C_VEL
LIN {X 0,Y 100.332,Z 382.302,A -85,B 0,C 180,E1 -27410.919,E2 -27410.919} C_VEL
LIN {X 0,Y 96.57,Z 384.592,A -85,B 0,C 180,E1 -27414.395,E2 -27414.395} C_VEL
LIN {X 0,Y 93.265,Z 386.466,A -85,B 0,C 180,E1 -27418.165,E2 -27418.165} C_VEL
LIN {X 0,Y 87.952,Z 388.942,A -85,B 0,C 180,E1 -27426.452,E2 -27426.452} C_VEL
LIN {X 0,Y 84.915,Z 389.921,A -85,B 0,C 180,E1 -27435.624,E2 -27435.624} C_VEL
LIN {X 0,Y 84.124,Z 389.816,A -85,B 0,C 180,E1 -27440.383,E2 -27440.383} C_VEL
LIN {X 0,Y 83.854,Z 389.315,A -85,B 0,C 180,E1 -27445.193,E2 -27445.193} C_VEL
LIN {X 0,Y 84.02,Z 388.43,A -85,B 0,C 180,E1 -27450.001,E2 -27450.001} C_VEL
LIN {X 0,Y 83.869,Z 387.102,A -85,B 0,C 180,E1 -27454.808,E2 -27454.808} C_VEL
LIN {X 0,Y 84.51,Z 384.254,A -85,B 0,C 180,E1 -27462.001,E2 -27462.001} C_VEL
LIN {X 0,Y 86.13,Z 380.335,A -85,B 0,C 180,E1 -27469.051,E2 -27469.051} C_VEL
LIN {X 0,Y 88.948,Z 375.258,A -85,B 0,C 180,E1 -27475.759,E2 -27475.759} C_VEL
LIN {X 0,Y 92.842,Z 368.843,A -85,B 0,C 180,E1 -27481.999,E2 -27481.999} C_VEL
LIN {X 0,Y 97.273,Z 361.377,A -85,B 0,C 180,E1 -27487.363,E2 -27487.363} C_VEL
LIN {X 0,Y 102.357,Z 352.548,A -85,B 0,C 180,E1 -27492.026,E2 -27492.026} C_VEL
LIN {X 0,Y 107.634,Z 342.517,A -85,B 0,C 180,E1 -27495.912,E2 -27495.912} C_VEL
LIN {X 0,Y 112.82,Z 331.195,A -85,B 0,C 180,E1 -27499.054,E2 -27499.054} C_VEL
LIN {X 0,Y 117.046,Z 320.1,A -85,B 0,C 180,E1 -27501.315,E2 -27501.315} C_VEL
LIN {X 0,Y 120.595,Z 309.022,A -85,B 0,C 180,E1 -27502.91,E2 -27502.91} C_VEL
LIN {X 0,Y 123.624,Z 295.869,A -85,B 0,C 180,E1 -27504.287,E2 -27504.287} C_VEL
LIN {X 0,Y 125.612,Z 282.066,A -85,B 0,C 180,E1 -27505.194,E2 -27505.194} C_VEL
LIN {X 0,Y 128.047,Z 254.068,A -85,B 0,C 180,E1 -27506.473,E2 -27506.473} C_VEL
LIN {X 0,Y 126.79,Z 249.802,A -85,B 0,C 180,E1 -27507.498,E2 -27507.498} C_VEL
LIN {X 0,Y 124.908,Z 245.194,A -85,B 0,C 180,E1 -27508.947,E2 -27508.947} C_VEL
LIN {X 0,Y 121.561,Z 240.321,A -85,B 0,C 180,E1 -27511.414,E2 -27511.414} C_VEL
LIN {X 0,Y 113.667,Z 231.18,A -85,B 0,C 180,E1 -27518.165,E2 -27518.165} C_VEL
LIN {X 0,Y 109.959,Z 224.985,A -85,B 0,C 180,E1 -27522.502,E2 -27522.502} C_VEL
LIN {X 0,Y 107.41,Z 221.043,A -85,B 0,C 180,E1 -27525.97,E2 -27525.97} C_VEL
LIN {X 0,Y 105.034,Z 217.24,A -85,B 0,C 180,E1 -27529.926,E2 -27529.926} C_VEL
LIN {X 0,Y 102.429,Z 213.296,A -85,B 0,C 180,E1 -27535.457,E2 -27535.457} C_VEL
LIN {X 0,Y 102.063,Z 212.355,A -85,B 0,C 180,E1 -27536.543,E2 -27536.543} C_VEL
LIN {X 0,Y 100.146,Z 210.54,A -85,B 0,C 180,E1 -27543.014,E2 -27543.014} C_VEL
LIN {X 0,Y 99.398,Z 209.779,A -85,B 0,C 180,E1 -27548.152,E2 -27548.152} C_VEL
LIN {X 0,Y 99.312,Z 210.06,A -85,B 0,C 180,E1 -27553.706,E2 -27553.706} C_VEL
LIN {X 0,Y 101.849,Z 212.769,A -85,B 0,C 180,E1 -27565.695,E2 -27565.695} C_VEL
LIN {X 0,Y 103.623,Z 216.066,A -85,B 0,C 180,E1 -27570.156,E2 -27570.156} C_VEL
LIN {X 0,Y 105.26,Z 217.944,A -85,B 0,C 180,E1 -27573.159,E2 -27573.159} C_VEL
LIN {X 0,Y 108.084,Z 222.255,A -85,B 0,C 180,E1 -27577.651,E2 -27577.651} C_VEL
LIN {X 0,Y 111.478,Z 227.608,A -85,B 0,C 180,E1 -27581.987,E2 -27581.987} C_VEL
LIN {X 0,Y 115.602,Z 234.683,A -85,B 0,C 180,E1 -27586.446,E2 -27586.446} C_VEL
LIN {X 0,Y 120.213,Z 243.789,A -85,B 0,C 180,E1 -27590.696,E2 -27590.696} C_VEL
LIN {X 0,Y 123.547,Z 251.363,A -85,B 0,C 180,E1 -27593.487,E2 -27593.487} C_VEL
LIN {X 0,Y 120.557,Z 281.313,A -85,B 0,C 180,E1 -27594.855,E2 -27594.855} C_VEL
LIN {X 0,Y 118.166,Z 294.672,A -85,B 0,C 180,E1 -27595.947,E2 -27595.947} C_VEL
LIN {X 0,Y 115.131,Z 306.692,A -85,B 0,C 180,E1 -27597.455,E2 -27597.455} C_VEL
LIN {X 0,Y 111.056,Z 318.795,A -85,B 0,C 180,E1 -27599.583,E2 -27599.583} C_VEL
LIN {X 0,Y 106.211,Z 330.426,A -85,B 0,C 180,E1 -27602.406,E2 -27602.406} C_VEL
LIN {X 0,Y 100.859,Z 341.099,A -85,B 0,C 180,E1 -27605.933,E2 -27605.933} C_VEL
LIN {X 0,Y 96.148,Z 349.461,A -85,B 0,C 180,E1 -27609.682,E2 -27609.682} C_VEL
LIN {X 0,Y 90.334,Z 358.753,A -85,B 0,C 180,E1 -27615.353,E2 -27615.353} C_VEL
LIN {X 0,Y 86.149,Z 365.057,A -85,B 0,C 180,E1 -27620.609,E2 -27620.609} C_VEL
LIN {X 0,Y 81.999,Z 371.239,A -85,B 0,C 180,E1 -27627.543,E2 -27627.543} C_VEL
LIN {X 0,Y 79.004,Z 376.084,A -85,B 0,C 180,E1 -27635.103,E2 -27635.103} C_VEL
LIN {X 0,Y 77.074,Z 379.764,A -85,B 0,C 180,E1 -27643.176,E2 -27643.176} C_VEL
LIN {X 0,Y 76.441,Z 382.708,A -85,B 0,C 180,E1 -27653.173,E2 -27653.173} C_VEL
LIN {X 0,Y 77.588,Z 384.203,A -85,B 0,C 180,E1 -27662.92,E2 -27662.92} C_VEL
LIN {X 0,Y 79.132,Z 384.444,A -85,B 0,C 180,E1 -27668.439,E2 -27668.439} C_VEL
LIN {X 0,Y 83.33,Z 383.725,A -85,B 0,C 180,E1 -27677.574,E2 -27677.574} C_VEL
LIN {X 0,Y 87.403,Z 382.346,A -85,B 0,C 180,E1 -27683.522,E2 -27683.522} C_VEL
LIN {X 0,Y 93.355,Z 379.642,A -85,B 0,C 180,E1 -27689.967,E2 -27689.967} C_VEL
LIN {X 0,Y 100.309,Z 375.73,A -85,B 0,C 180,E1 -27695.619,E2 -27695.619} C_VEL
LIN {X 0,Y 107.533,Z 370.905,A -85,B 0,C 180,E1 -27700.167,E2 -27700.167} C_VEL
LIN {X 0,Y 115.144,Z 364.961,A -85,B 0,C 180,E1 -27704.012,E2 -27704.012} C_VEL
LIN {X 0,Y 122.563,Z 358.214,A -85,B 0,C 180,E1 -27707.112,E2 -27707.112} C_VEL
LIN {X 0,Y 130.051,Z 350.219,A -85,B 0,C 180,E1 -27709.817,E2 -27709.817} C_VEL
LIN {X 0,Y 137.467,Z 340.807,A -85,B 0,C 180,E1 -27712.114,E2 -27712.114} C_VEL
LIN {X 0,Y 144.204,Z 330.526,A -85,B 0,C 180,E1 -27713.931,E2 -27713.931} C_VEL
LIN {X 0,Y 149.836,Z 319.998,A -85,B 0,C 180,E1 -27715.358,E2 -27715.358} C_VEL
LIN {X 0,Y 154.897,Z 308.134,A -85,B 0,C 180,E1 -27716.548,E2 -27716.548} C_VEL
LIN {X 0,Y 158.87,Z 295.51,A -85,B 0,C 180,E1 -27717.467,E2 -27717.467} C_VEL
LIN {X 0,Y 161.734,Z 282.322,A -85,B 0,C 180,E1 -27718.08,E2 -27718.08} C_VEL
LIN {X 0,Y 162.31,Z 278.203,A -85,B 0,C 180,E1 -27718.264,E2 -27718.264} C_VEL
LIN {X 0,Y 160.945,Z 274.164,A -85,B 0,C 180,E1 -27721.517,E2 -27721.517} C_VEL
LIN {X 0,Y 160.045,Z 271.408,A -85,B 0,C 180,E1 -27724.409,E2 -27724.409} C_VEL
LIN {X 0,Y 159.288,Z 268.81,A -85,B 0,C 180,E1 -27730.482,E2 -27730.482} C_VEL
LIN {X 0,Y 160.185,Z 272.673,A -85,B 0,C 180,E1 -27737.888,E2 -27737.888} C_VEL
LIN {X 0,Y 161.029,Z 275.255,A -85,B 0,C 180,E1 -27740.438,E2 -27740.438} C_VEL
LIN {X 0,Y 162.166,Z 280.161,A -85,B 0,C 180,E1 -27743.378,E2 -27743.378} C_VEL
LIN {X 0,Y 160.115,Z 292.104,A -85,B 0,C 180,E1 -27743.861,E2 -27743.861} C_VEL
LIN {X 0,Y 156.843,Z 304.248,A -85,B 0,C 180,E1 -27744.479,E2 -27744.479} C_VEL
LIN {X 0,Y 152.504,Z 315.931,A -85,B 0,C 180,E1 -27745.258,E2 -27745.258} C_VEL
LIN {X 0,Y 147.07,Z 327.325,A -85,B 0,C 180,E1 -27746.363,E2 -27746.363} C_VEL
LIN {X 0,Y 140.183,Z 338.865,A -85,B 0,C 180,E1 -27747.918,E2 -27747.918} C_VEL
LIN {X 0,Y 133.548,Z 348.185,A -85,B 0,C 180,E1 -27749.737,E2 -27749.737} C_VEL
LIN {X 0,Y 126.284,Z 356.766,A -85,B 0,C 180,E1 -27751.93,E2 -27751.93} C_VEL
LIN {X 0,Y 117.894,Z 365.164,A -85,B 0,C 180,E1 -27754.948,E2 -27754.948} C_VEL
LIN {X 0,Y 108.684,Z 372.967,A -85,B 0,C 180,E1 -27759.107,E2 -27759.107} C_VEL
LIN {X 0,Y 101.447,Z 378.255,A -85,B 0,C 180,E1 -27763.331,E2 -27763.331} C_VEL
LIN {X 0,Y 94.916,Z 382.417,A -85,B 0,C 180,E1 -27768.211,E2 -27768.211} C_VEL
LIN {X 0,Y 90.892,Z 384.651,A -85,B 0,C 180,E1 -27771.788,E2 -27771.788} C_VEL
LIN {X 0,Y 84.142,Z 387.799,A -85,B 0,C 180,E1 -27779.925,E2 -27779.925} C_VEL
LIN {X 0,Y 79.469,Z 389.423,A -85,B 0,C 180,E1 -27789.284,E2 -27789.284} C_VEL
LIN {X 0,Y 78.022,Z 389.657,A -85,B 0,C 180,E1 -27794.323,E2 -27794.323} C_VEL
LIN {X 0,Y 76.774,Z 388.942,A -85,B 0,C 180,E1 -27804.749,E2 -27804.749} C_VEL
LIN {X 0,Y 76.917,Z 388.012,A -85,B 0,C 180,E1 -27810.001,E2 -27810.001} C_VEL
LIN {X 0,Y 76.789,Z 386.627,A -85,B 0,C 180,E1 -27815.252,E2 -27815.252} C_VEL
LIN {X 0,Y 77.561,Z 383.69,A -85,B 0,C 180,E1 -27823.094,E2 -27823.094} C_VEL
LIN {X 0,Y 79.413,Z 379.666,A -85,B 0,C 180,E1 -27830.733,E2 -27830.733} C_VEL
LIN {X 0,Y 83.246,Z 373.45,A -85,B 0,C 180,E1 -27839.043,E2 -27839.043} C_VEL
LIN {X 0,Y 87.713,Z 366.644,A -85,B 0,C 180,E1 -27845.515,E2 -27845.515} C_VEL
LIN {X 0,Y 91.231,Z 361.016,A -85,B 0,C 180,E1 -27849.609,E2 -27849.609} C_VEL
LIN {X 0,Y 97.173,Z 351.279,A -85,B 0,C 180,E1 -27854.845,E2 -27854.845} C_VEL
LIN {X 0,Y 102.826,Z 340.973,A -85,B 0,C 180,E1 -27858.751,E2 -27858.751} C_VEL
LIN {X 0,Y 107.637,Z 330.75,A -85,B 0,C 180,E1 -27861.586,E2 -27861.586} C_VEL
LIN {X 0,Y 112.073,Z 319.618,A -85,B 0,C 180,E1 -27863.843,E2 -27863.843} C_VEL
LIN {X 0,Y 115.764,Z 308.478,A -85,B 0,C 180,E1 -27865.426,E2 -27865.426} C_VEL
LIN {X 0,Y 118.861,Z 295.492,A -85,B 0,C 180,E1 -27866.764,E2 -27866.764} C_VEL
LIN {X 0,Y 120.878,Z 282.108,A -85,B 0,C 180,E1 -27867.638,E2 -27867.638} C_VEL
LIN {X 0,Y 123.28,Z 256.537,A -85,B 0,C 180,E1 -27868.775,E2 -27868.775} C_VEL
LIN {X 0,Y 121.519,Z 250.142,A -85,B 0,C 180,E1 -27870.433,E2 -27870.433} C_VEL
LIN {X 0,Y 117.329,Z 238.106,A -85,B 0,C 180,E1 -27874.489,E2 -27874.489} C_VEL
LIN {X 0,Y 113.667,Z 231.18,A -85,B 0,C 180,E1 -27878.165,E2 -27878.165} C_VEL
LIN {X 0,Y 111.392,Z 228.491,A -85,B 0,C 180,E1 -27880.576,E2 -27880.576} C_VEL
LIN {X 0,Y 108.996,Z 226.72,A -85,B 0,C 180,E1 -27883.245,E2 -27883.245} C_VEL
LIN {X 0,Y 103.368,Z 223.528,A -85,B 0,C 180,E1 -27891.179,E2 -27891.179} C_VEL
LIN {X 0,Y 102.308,Z 222.417,A -85,B 0,C 180,E1 -27893.248,E2 -27893.248} C_VEL
LIN {X 0,Y 100.521,Z 219.016,A -85,B 0,C 180,E1 -27898.119,E2 -27898.119} C_VEL
LIN {X 0,Y 99.204,Z 217.57,A -85,B 0,C 180,E1 -27903.042,E2 -27903.042} C_VEL
LIN {X 0,Y 98.464,Z 216.827,A -85,B 0,C 180,E1 -27908.204,E2 -27908.204} C_VEL
LIN {X 0,Y 98.385,Z 217.151,A -85,B 0,C 180,E1 -27913.837,E2 -27913.837} C_VEL
LIN {X 0,Y 100.552,Z 219.677,A -85,B 0,C 180,E1 -27924.791,E2 -27924.791} C_VEL
LIN {X 0,Y 102.44,Z 223.143,A -85,B 0,C 180,E1 -27929.795,E2 -27929.795} C_VEL
LIN {X 0,Y 103.518,Z 224.495,A -85,B 0,C 180,E1 -27931.905,E2 -27931.905} C_VEL
LIN {X 0,Y 106,Z 228.541,A -85,B 0,C 180,E1 -27936.223,E2 -27936.223} C_VEL
LIN {X 0,Y 109.067,Z 233.66,A -85,B 0,C 180,E1 -27940.52,E2 -27940.52} C_VEL
LIN {X 0,Y 112.761,Z 240.398,A -85,B 0,C 180,E1 -27944.871,E2 -27944.871} C_VEL
LIN {X 0,Y 116.902,Z 249.154,A -85,B 0,C 180,E1 -27949.071,E2 -27949.071} C_VEL
LIN {X 0,Y 118.934,Z 253.863,A -85,B 0,C 180,E1 -27950.932,E2 -27950.932} C_VEL
LIN {X 0,Y 116.066,Z 281.508,A -85,B 0,C 180,E1 -27952.201,E2 -27952.201} C_VEL
LIN {X 0,Y 113.477,Z 295.342,A -85,B 0,C 180,E1 -27953.328,E2 -27953.328} C_VEL
LIN {X 0,Y 110.083,Z 307.908,A -85,B 0,C 180,E1 -27954.928,E2 -27954.928} C_VEL
LIN {X 0,Y 105.516,Z 320.598,A -85,B 0,C 180,E1 -27957.235,E2 -27957.235} C_VEL
LIN {X 0,Y 100.402,Z 331.955,A -85,B 0,C 180,E1 -27960.082,E2 -27960.082} C_VEL
LIN {X 0,Y 94.932,Z 342.144,A -85,B 0,C 180,E1 -27963.627,E2 -27963.627} C_VEL
LIN {X 0,Y 89.307,Z 351.38,A -85,B 0,C 180,E1 -27968.049,E2 -27968.049} C_VEL
LIN {X 0,Y 84.202,Z 358.985,A -85,B 0,C 180,E1 -27973.013,E2 -27973.013} C_VEL
LIN {X 0,Y 78.889,Z 366.444,A -85,B 0,C 180,E1 -27979.735,E2 -27979.735} C_VEL
LIN {X 0,Y 74.609,Z 372.357,A -85,B 0,C 180,E1 -27987.299,E2 -27987.299} C_VEL
LIN {X 0,Y 71.569,Z 376.993,A -85,B 0,C 180,E1 -27995.634,E2 -27995.634} C_VEL
LIN {X 0,Y 70.208,Z 379.456,A -85,B 0,C 180,E1 -28001.548,E2 -28001.548} C_VEL
LIN {X 0,Y 69.421,Z 381.445,A -85,B 0,C 180,E1 -28007.679,E2 -28007.679} C_VEL
LIN {X 0,Y 69.363,Z 382.991,A -85,B 0,C 180,E1 -28014.244,E2 -28014.244} C_VEL
LIN {X 0,Y 69.9,Z 383.981,A -85,B 0,C 180,E1 -28020.179,E2 -28020.179} C_VEL
LIN {X 0,Y 71.857,Z 384.659,A -85,B 0,C 180,E1 -28028.523,E2 -28028.523} C_VEL
LIN {X 0,Y 75.834,Z 384.362,A -85,B 0,C 180,E1 -28037.85,E2 -28037.85} C_VEL
LIN {X 0,Y 79.122,Z 383.555,A -85,B 0,C 180,E1 -28043.074,E2 -28043.074} C_VEL
LIN {X 0,Y 85.343,Z 381.319,A -85,B 0,C 180,E1 -28050.394,E2 -28050.394} C_VEL
LIN {X 0,Y 92.126,Z 378.147,A -85,B 0,C 180,E1 -28056.267,E2 -28056.267} C_VEL
LIN {X 0,Y 100.063,Z 373.616,A -85,B 0,C 180,E1 -28061.473,E2 -28061.473} C_VEL
LIN {X 0,Y 108.71,Z 367.691,A -85,B 0,C 180,E1 -28065.865,E2 -28065.865} C_VEL
LIN {X 0,Y 116.515,Z 361.33,A -85,B 0,C 180,E1 -28069.095,E2 -28069.095} C_VEL
LIN {X 0,Y 124.262,Z 353.904,A -85,B 0,C 180,E1 -28071.792,E2 -28071.792} C_VEL
LIN {X 0,Y 131.978,Z 345.1,A -85,B 0,C 180,E1 -28074.117,E2 -28074.117} C_VEL
LIN {X 0,Y 139.147,Z 335.336,A -85,B 0,C 180,E1 -28075.968,E2 -28075.968} C_VEL
LIN {X 0,Y 145.975,Z 323.993,A -85,B 0,C 180,E1 -28077.562,E2 -28077.562} C_VEL
LIN {X 0,Y 151.574,Z 312.146,A -85,B 0,C 180,E1 -28078.794,E2 -28078.794} C_VEL
LIN {X 0,Y 156.147,Z 299.424,A -85,B 0,C 180,E1 -28079.745,E2 -28079.745} C_VEL
LIN {X 0,Y 159.333,Z 286.951,A -85,B 0,C 180,E1 -28080.379,E2 -28080.379} C_VEL
LIN {X 0,Y 160.104,Z 282.73,A -85,B 0,C 180,E1 -28080.552,E2 -28080.552} C_VEL
LIN {X 0,Y 159.274,Z 279.818,A -85,B 0,C 180,E1 -28083.322,E2 -28083.322} C_VEL
LIN {X 0,Y 158.825,Z 278.066,A -85,B 0,C 180,E1 -28085.398,E2 -28085.398} C_VEL
LIN {X 0,Y 158.365,Z 275.884,A -85,B 0,C 180,E1 -28090.227,E2 -28090.227} C_VEL
LIN {X 0,Y 159.03,Z 279.552,A -85,B 0,C 180,E1 -28097.358,E2 -28097.358} C_VEL
LIN {X 0,Y 159.618,Z 281.773,A -85,B 0,C 180,E1 -28099.535,E2 -28099.535} C_VEL
LIN {X 0,Y 160.026,Z 284.124,A -85,B 0,C 180,E1 -28101.055,E2 -28101.055} C_VEL
LIN {X 0,Y 157.203,Z 297.094,A -85,B 0,C 180,E1 -28101.591,E2 -28101.591} C_VEL
LIN {X 0,Y 153.082,Z 309.845,A -85,B 0,C 180,E1 -28102.281,E2 -28102.281} C_VEL
LIN {X 0,Y 148.071,Z 321.408,A -85,B 0,C 180,E1 -28103.132,E2 -28103.132} C_VEL
LIN {X 0,Y 141.727,Z 332.913,A -85,B 0,C 180,E1 -28104.331,E2 -28104.331} C_VEL
LIN {X 0,Y 134.732,Z 343.297,A -85,B 0,C 180,E1 -28105.868,E2 -28105.868} C_VEL
LIN {X 0,Y 127.208,Z 352.686,A -85,B 0,C 180,E1 -28107.876,E2 -28107.876} C_VEL
LIN {X 0,Y 119.802,Z 360.447,A -85,B 0,C 180,E1 -28110.086,E2 -28110.086} C_VEL
LIN {X 0,Y 111.186,Z 368.089,A -85,B 0,C 180,E1 -28113.121,E2 -28113.121} C_VEL
LIN {X 0,Y 101.721,Z 375.167,A -85,B 0,C 180,E1 -28117.389,E2 -28117.389} C_VEL
LIN {X 0,Y 94.321,Z 379.927,A -85,B 0,C 180,E1 -28121.832,E2 -28121.832} C_VEL
LIN {X 0,Y 87.543,Z 383.638,A -85,B 0,C 180,E1 -28126.971,E2 -28126.971} C_VEL
LIN {X 0,Y 81.493,Z 386.383,A -85,B 0,C 180,E1 -28132.867,E2 -28132.867} C_VEL
LIN {X 0,Y 75.096,Z 388.656,A -85,B 0,C 180,E1 -28142.101,E2 -28142.101} C_VEL
LIN {X 0,Y 72.827,Z 389.215,A -85,B 0,C 180,E1 -28147.295,E2 -28147.295} C_VEL
LIN {X 0,Y 70.133,Z 389.156,A -85,B 0,C 180,E1 -28158.44,E2 -28158.44} C_VEL
LIN {X 0,Y 69.715,Z 388.568,A -85,B 0,C 180,E1 -28164.215,E2 -28164.215} C_VEL
LIN {X 0,Y 69.822,Z 387.594,A -85,B 0,C 180,E1 -28170.001,E2 -28170.001} C_VEL
LIN {X 0,Y 69.732,Z 386.12,A -85,B 0,C 180,E1 -28175.786,E2 -28175.786} C_VEL
LIN {X 0,Y 70.622,Z 383.088,A -85,B 0,C 180,E1 -28184.407,E2 -28184.407} C_VEL
LIN {X 0,Y 72.762,Z 378.957,A -85,B 0,C 180,E1 -28192.729,E2 -28192.729} C_VEL
LIN {X 0,Y 77.073,Z 372.617,A -85,B 0,C 180,E1 -28201.624,E2 -28201.624} C_VEL
LIN {X 0,Y 81.868,Z 365.807,A -85,B 0,C 180,E1 -28208.329,E2 -28208.329} C_VEL
LIN {X 0,Y 86.587,Z 358.872,A -85,B 0,C 180,E1 -28213.305,E2 -28213.305} C_VEL
LIN {X 0,Y 92.238,Z 349.982,A -85,B 0,C 180,E1 -28217.98,E2 -28217.98} C_VEL
LIN {X 0,Y 97.64,Z 340.565,A -85,B 0,C 180,E1 -28221.516,E2 -28221.516} C_VEL
LIN {X 0,Y 102.702,Z 330.313,A -85,B 0,C 180,E1 -28224.354,E2 -28224.354} C_VEL
LIN {X 0,Y 107.338,Z 319.136,A -85,B 0,C 180,E1 -28226.598,E2 -28226.598} C_VEL
LIN {X 0,Y 111.171,Z 307.932,A -85,B 0,C 180,E1 -28228.158,E2 -28228.158} C_VEL
LIN {X 0,Y 114.354,Z 294.947,A -85,B 0,C 180,E1 -28229.464,E2 -28229.464} C_VEL
LIN {X 0,Y 116.412,Z 281.734,A -85,B 0,C 180,E1 -28230.309,E2 -28230.309} C_VEL
LIN {X 0,Y 118.72,Z 258.18,A -85,B 0,C 180,E1 -28231.351,E2 -28231.351} C_VEL
LIN {X 0,Y 115.281,Z 246.862,A -85,B 0,C 180,E1 -28234.964,E2 -28234.964} C_VEL
LIN {X 0,Y 113.516,Z 242.053,A -85,B 0,C 180,E1 -28236.905,E2 -28236.905} C_VEL
LIN {X 0,Y 109.615,Z 234.406,A -85,B 0,C 180,E1 -28241.447,E2 -28241.447} C_VEL
LIN {X 0,Y 106.793,Z 229.797,A -85,B 0,C 180,E1 -28245.197,E2 -28245.197} C_VEL
LIN {X 0,Y 105.163,Z 227.053,A -85,B 0,C 180,E1 -28247.755,E2 -28247.755} C_VEL
LIN {X 0,Y 102.842,Z 223.105,A -85,B 0,C 180,E1 -28252.141,E2 -28252.141} C_VEL
LIN {X 0,Y 102.308,Z 222.417,A -85,B 0,C 180,E1 -28253.248,E2 -28253.248} C_VEL
LIN {X 0,Y 100.904,Z 221.312,A -85,B 0,C 180,E1 -28256.423,E2 -28256.423} C_VEL
LIN {X 0,Y 99.629,Z 221.399,A -85,B 0,C 180,E1 -28259.747,E2 -28259.747} C_VEL
LIN {X 0,Y 97.501,Z 223.703,A -85,B 0,C 180,E1 -28268.998,E2 -28268.998} C_VEL
LIN {X 0,Y 97.403,Z 223.941,A -85,B 0,C 180,E1 -28271.382,E2 -28271.382} C_VEL
LIN {X 0,Y 99.174,Z 226.281,A -85,B 0,C 180,E1 -28283.442,E2 -28283.442} C_VEL
LIN {X 0,Y 101.117,Z 230.026,A -85,B 0,C 180,E1 -28289.108,E2 -28289.108} C_VEL
LIN {X 0,Y 102.026,Z 231.441,A -85,B 0,C 180,E1 -28291.06,E2 -28291.06} C_VEL
LIN {X 0,Y 104.092,Z 235.038,A -85,B 0,C 180,E1 -28294.931,E2 -28294.931} C_VEL
LIN {X 0,Y 107.066,Z 240.292,A -85,B 0,C 180,E1 -28299.451,E2 -28299.451} C_VEL
LIN {X 0,Y 110.674,Z 247.627,A -85,B 0,C 180,E1 -28304.023,E2 -28304.023} C_VEL
LIN {X 0,Y 113.919,Z 255.19,A -85,B 0,C 180,E1 -28307.617,E2 -28307.617} C_VEL
LIN {X 0,Y 114.505,Z 256.584,A -85,B 0,C 180,E1 -28308.214,E2 -28308.214} C_VEL
LIN {X 0,Y 111.886,Z 281.094,A -85,B 0,C 180,E1 -28309.325,E2 -28309.325} C_VEL
LIN {X 0,Y 109.222,Z 294.933,A -85,B 0,C 180,E1 -28310.398,E2 -28310.398} C_VEL
LIN {X 0,Y 105.616,Z 307.926,A -85,B 0,C 180,E1 -28312.009,E2 -28312.009} C_VEL
LIN {X 0,Y 101.475,Z 319.067,A -85,B 0,C 180,E1 -28313.934,E2 -28313.934} C_VEL
LIN {X 0,Y 96.14,Z 330.734,A -85,B 0,C 180,E1 -28316.751,E2 -28316.751} C_VEL
LIN {X 0,Y 90.312,Z 341.267,A -85,B 0,C 180,E1 -28320.257,E2 -28320.257} C_VEL
LIN {X 0,Y 84.72,Z 350.061,A -85,B 0,C 180,E1 -28324.351,E2 -28324.351} C_VEL
LIN {X 0,Y 78.225,Z 359.159,A -85,B 0,C 180,E1 -28330.31,E2 -28330.31} C_VEL
LIN {X 0,Y 72.538,Z 366.6,A -85,B 0,C 180,E1 -28337.361,E2 -28337.361} C_VEL
LIN {X 0,Y 68.547,Z 371.677,A -85,B 0,C 180,E1 -28344.114,E2 -28344.114} C_VEL
LIN {X 0,Y 65.014,Z 376.546,A -85,B 0,C 180,E1 -28353.097,E2 -28353.097} C_VEL
LIN {X 0,Y 62.803,Z 380.249,A -85,B 0,C 180,E1 -28362.932,E2 -28362.932} C_VEL
LIN {X 0,Y 62.315,Z 383.271,A -85,B 0,C 180,E1 -28375.558,E2 -28375.558} C_VEL
LIN {X 0,Y 63.333,Z 384.439,A -85,B 0,C 180,E1 -28383.699,E2 -28383.699} C_VEL
LIN {X 0,Y 65.379,Z 384.928,A -85,B 0,C 180,E1 -28391.203,E2 -28391.203} C_VEL
LIN {X 0,Y 67.609,Z 384.927,A -85,B 0,C 180,E1 -28396.689,E2 -28396.689} C_VEL
LIN {X 0,Y 71.762,Z 384.275,A -85,B 0,C 180,E1 -28404.019,E2 -28404.019} C_VEL
LIN {X 0,Y 79.073,Z 382.17,A -85,B 0,C 180,E1 -28412.722,E2 -28412.722} C_VEL
LIN {X 0,Y 86.545,Z 379.124,A -85,B 0,C 180,E1 -28419.044,E2 -28419.044} C_VEL
LIN {X 0,Y 94.91,Z 374.827,A -85,B 0,C 180,E1 -28424.286,E2 -28424.286} C_VEL
LIN {X 0,Y 104.638,Z 368.657,A -85,B 0,C 180,E1 -28428.936,E2 -28428.936} C_VEL
LIN {X 0,Y 113.471,Z 361.878,A -85,B 0,C 180,E1 -28432.298,E2 -28432.298} C_VEL
LIN {X 0,Y 121.714,Z 354.351,A -85,B 0,C 180,E1 -28434.899,E2 -28434.899} C_VEL
LIN {X 0,Y 130.59,Z 344.538,A -85,B 0,C 180,E1 -28437.282,E2 -28437.282} C_VEL
LIN {X 0,Y 137.946,Z 334.702,A -85,B 0,C 180,E1 -28438.962,E2 -28438.962} C_VEL
LIN {X 0,Y 144.472,Z 324.047,A -85,B 0,C 180,E1 -28440.319,E2 -28440.319} C_VEL
LIN {X 0,Y 150.094,Z 312.417,A -85,B 0,C 180,E1 -28441.435,E2 -28441.435} C_VEL
LIN {X 0,Y 154.741,Z 299.812,A -85,B 0,C 180,E1 -28442.306,E2 -28442.306} C_VEL
LIN {X 0,Y 157.968,Z 287.44,A -85,B 0,C 180,E1 -28442.951,E2 -28442.951} C_VEL
LIN {X 0,Y 157.484,Z 284.771,A -85,B 0,C 180,E1 -28446.086,E2 -28446.086} C_VEL
LIN {X 0,Y 157.273,Z 283.001,A -85,B 0,C 180,E1 -28450.299,E2 -28450.299} C_VEL
LIN {X 0,Y 157.663,Z 286.553,A -85,B 0,C 180,E1 -28457.012,E2 -28457.012} C_VEL
LIN {X 0,Y 157.983,Z 288.248,A -85,B 0,C 180,E1 -28458.669,E2 -28458.669} C_VEL
LIN {X 0,Y 154.584,Z 301.423,A -85,B 0,C 180,E1 -28459.237,E2 -28459.237} C_VEL
LIN {X 0,Y 149.533,Z 314.864,A -85,B 0,C 180,E1 -28459.95,E2 -28459.95} C_VEL
LIN {X 0,Y 143.839,Z 326.381,A -85,B 0,C 180,E1 -28460.861,E2 -28460.861} C_VEL
LIN {X 0,Y 136.567,Z 337.981,A -85,B 0,C 180,E1 -28462.133,E2 -28462.133} C_VEL
LIN {X 0,Y 128.692,Z 348.307,A -85,B 0,C 180,E1 -28463.832,E2 -28463.832} C_VEL
LIN {X 0,Y 120.981,Z 356.736,A -85,B 0,C 180,E1 -28465.788,E2 -28465.788} C_VEL
LIN {X 0,Y 111.921,Z 365.015,A -85,B 0,C 180,E1 -28468.464,E2 -28468.464} C_VEL
LIN {X 0,Y 103.168,Z 371.737,A -85,B 0,C 180,E1 -28471.623,E2 -28471.623} C_VEL
LIN {X 0,Y 94.885,Z 377.148,A -85,B 0,C 180,E1 -28475.438,E2 -28475.438} C_VEL
LIN {X 0,Y 86.759,Z 381.672,A -85,B 0,C 180,E1 -28480.399,E2 -28480.399} C_VEL
LIN {X 0,Y 80.217,Z 384.694,A -85,B 0,C 180,E1 -28485.502,E2 -28485.502} C_VEL
LIN {X 0,Y 72.172,Z 387.62,A -85,B 0,C 180,E1 -28494.25,E2 -28494.25} C_VEL
LIN {X 0,Y 68.883,Z 388.501,A -85,B 0,C 180,E1 -28499.328,E2 -28499.328} C_VEL
LIN {X 0,Y 64.422,Z 389.086,A -85,B 0,C 180,E1 -28510.898,E2 -28510.898} C_VEL
LIN {X 0,Y 62.639,Z 388.186,A -85,B 0,C 180,E1 -28523.559,E2 -28523.559} C_VEL
LIN {X 0,Y 62.718,Z 387.129,A -85,B 0,C 180,E1 -28530.001,E2 -28530.001} C_VEL
LIN {X 0,Y 62.657,Z 385.589,A -85,B 0,C 180,E1 -28536.442,E2 -28536.442} C_VEL
LIN {X 0,Y 63.743,Z 382.454,A -85,B 0,C 180,E1 -28546.001,E2 -28546.001} C_VEL
LIN {X 0,Y 66.224,Z 378.21,A -85,B 0,C 180,E1 -28555.121,E2 -28555.121} C_VEL
LIN {X 0,Y 71.092,Z 371.754,A -85,B 0,C 180,E1 -28564.642,E2 -28564.642} C_VEL
LIN {X 0,Y 76.736,Z 364.174,A -85,B 0,C 180,E1 -28572.193,E2 -28572.193} C_VEL
LIN {X 0,Y 82.893,Z 355.737,A -85,B 0,C 180,E1 -28577.89,E2 -28577.89} C_VEL
LIN {X 0,Y 88.87,Z 346.598,A -85,B 0,C 180,E1 -28582.264,E2 -28582.264} C_VEL
LIN {X 0,Y 94.671,Z 336.513,A -85,B 0,C 180,E1 -28585.679,E2 -28585.679} C_VEL
LIN {X 0,Y 100.097,Z 325.31,A -85,B 0,C 180,E1 -28588.358,E2 -28588.358} C_VEL
LIN {X 0,Y 104.334,Z 314.782,A -85,B 0,C 180,E1 -28590.145,E2 -28590.145} C_VEL
LIN {X 0,Y 108.293,Z 302.182,A -85,B 0,C 180,E1 -28591.666,E2 -28591.666} C_VEL
LIN {X 0,Y 111.103,Z 289.141,A -85,B 0,C 180,E1 -28592.728,E2 -28592.728} C_VEL
LIN {X 0,Y 113.245,Z 271.281,A -85,B 0,C 180,E1 -28593.612,E2 -28593.612} C_VEL
LIN {X 0,Y 114.324,Z 260.106,A -85,B 0,C 180,E1 -28594.124,E2 -28594.124} C_VEL
LIN {X 0,Y 111.004,Z 248.608,A -85,B 0,C 180,E1 -28598.16,E2 -28598.16} C_VEL
LIN {X 0,Y 107.974,Z 241.969,A -85,B 0,C 180,E1 -28601.963,E2 -28601.963} C_VEL
LIN {X 0,Y 105.08,Z 236.632,A -85,B 0,C 180,E1 -28606.082,E2 -28606.082} C_VEL
LIN {X 0,Y 103.185,Z 233.27,A -85,B 0,C 180,E1 -28609.325,E2 -28609.325} C_VEL
LIN {X 0,Y 101.154,Z 229.582,A -85,B 0,C 180,E1 -28613.558,E2 -28613.558} C_VEL
LIN {X 0,Y 99.324,Z 225.904,A -85,B 0,C 180,E1 -28618.856,E2 -28618.856} C_VEL
LIN {X 0,Y 98.048,Z 224.471,A -85,B 0,C 180,E1 -28624.107,E2 -28624.107} C_VEL
LIN {X 0,Y 97.527,Z 223.883,A -85,B 0,C 180,E1 -28628.283,E2 -28628.283} C_VEL
LIN {X 0,Y 97.403,Z 223.941,A -85,B 0,C 180,E1 -28631.382,E2 -28631.382} C_VEL
LIN {X 0,Y 97.396,Z 224.638,A -85,B 0,C 180,E1 -28633.652,E2 -28633.652} C_VEL
LIN {X 0,Y 97.382,Z 226.27,A -85,B 0,C 180,E1 -28635.783,E2 -28635.783} C_VEL
LIN {X 0,Y 97.813,Z 232.722,A -85,B 0,C 180,E1 -28641.899,E2 -28641.899} C_VEL
LIN {X 0,Y 97.97,Z 233.27,A -85,B 0,C 180,E1 -28642.626,E2 -28642.626} C_VEL
LIN {X 0,Y 100.289,Z 237.798,A -85,B 0,C 180,E1 -28649.559,E2 -28649.559} C_VEL
LIN {X 0,Y 102.353,Z 241.689,A -85,B 0,C 180,E1 -28653.794,E2 -28653.794} C_VEL
LIN {X 0,Y 104.729,Z 246.297,A -85,B 0,C 180,E1 -28657.798,E2 -28657.798} C_VEL
LIN {X 0,Y 107.823,Z 253.036,A -85,B 0,C 180,E1 -28662.141,E2 -28662.141} C_VEL
LIN {X 0,Y 110.415,Z 259.644,A -85,B 0,C 180,E1 -28665.391,E2 -28665.391} C_VEL
LIN {X 0,Y 107.701,Z 282.398,A -85,B 0,C 180,E1 -28666.327,E2 -28666.327} C_VEL
LIN {X 0,Y 104.987,Z 295.736,A -85,B 0,C 180,E1 -28667.365,E2 -28667.365} C_VEL
LIN {X 0,Y 101.447,Z 307.923,A -85,B 0,C 180,E1 -28668.841,E2 -28668.841} C_VEL
LIN {X 0,Y 97.113,Z 319.121,A -85,B 0,C 180,E1 -28670.71,E2 -28670.71} C_VEL
LIN {X 0,Y 91.51,Z 330.825,A -85,B 0,C 180,E1 -28673.472,E2 -28673.472} C_VEL
LIN {X 0,Y 85.362,Z 341.397,A -85,B 0,C 180,E1 -28676.943,E2 -28676.943} C_VEL
LIN {X 0,Y 78.466,Z 351.515,A -85,B 0,C 180,E1 -28681.804,E2 -28681.804} C_VEL
LIN {X 0,Y 72.445,Z 359.334,A -85,B 0,C 180,E1 -28687.166,E2 -28687.166} C_VEL
LIN {X 0,Y 66.639,Z 366.397,A -85,B 0,C 180,E1 -28694.127,E2 -28694.127} C_VEL
LIN {X 0,Y 61.204,Z 372.772,A -85,B 0,C 180,E1 -28703.405,E2 -28703.405} C_VEL
LIN {X 0,Y 57.535,Z 377.443,A -85,B 0,C 180,E1 -28713.5,E2 -28713.5} C_VEL
LIN {X 0,Y 55.44,Z 380.974,A -85,B 0,C 180,E1 -28724.685,E2 -28724.685} C_VEL
LIN {X 0,Y 55.308,Z 383.547,A -85,B 0,C 180,E1 -28737.205,E2 -28737.205} C_VEL
LIN {X 0,Y 57.056,Z 384.84,A -85,B 0,C 180,E1 -28748.015,E2 -28748.015} C_VEL
LIN {X 0,Y 59.386,Z 385.22,A -85,B 0,C 180,E1 -28755.238,E2 -28755.238} C_VEL
LIN {X 0,Y 62.487,Z 385.146,A -85,B 0,C 180,E1 -28761.932,E2 -28761.932} C_VEL
LIN {X 0,Y 66.448,Z 384.552,A -85,B 0,C 180,E1 -28768.08,E2 -28768.08} C_VEL
LIN {X 0,Y 70.804,Z 383.559,A -85,B 0,C 180,E1 -28773.294,E2 -28773.294} C_VEL
LIN {X 0,Y 76.131,Z 381.918,A -85,B 0,C 180,E1 -28778.335,E2 -28778.335} C_VEL
LIN {X 0,Y 84.051,Z 378.803,A -85,B 0,C 180,E1 -28784.064,E2 -28784.064} C_VEL
LIN {X 0,Y 93.088,Z 374.318,A -85,B 0,C 180,E1 -28788.953,E2 -28788.953} C_VEL
LIN {X 0,Y 102.358,Z 368.673,A -85,B 0,C 180,E1 -28792.814,E2 -28792.814} C_VEL
LIN {X 0,Y 111,Z 362.33,A -85,B 0,C 180,E1 -28795.717,E2 -28795.717} C_VEL
LIN {X 0,Y 119.54,Z 354.854,A -85,B 0,C 180,E1 -28798.118,E2 -28798.118} C_VEL
LIN {X 0,Y 128.522,Z 345.313,A -85,B 0,C 180,E1 -28800.258,E2 -28800.258} C_VEL
LIN {X 0,Y 136.236,Z 335.342,A -85,B 0,C 180,E1 -28801.832,E2 -28801.832} C_VEL
LIN {X 0,Y 143.409,Z 323.907,A -85,B 0,C 180,E1 -28803.156,E2 -28803.156} C_VEL
LIN {X 0,Y 149.063,Z 312.408,A -85,B 0,C 180,E1 -28804.141,E2 -28804.141} C_VEL
LIN {X 0,Y 153.832,Z 299.712,A -85,B 0,C 180,E1 -28804.937,E2 -28804.937} C_VEL
LIN {X 0,Y 155.891,Z 292.518,A -85,B 0,C 180,E1 -28805.31,E2 -28805.31} C_VEL
LIN {X 0,Y 155.779,Z 291.193,A -85,B 0,C 180,E1 -28807.339,E2 -28807.339} C_VEL
LIN {X 0,Y 155.75,Z 290.126,A -85,B 0,C 180,E1 -28810.401,E2 -28810.401} C_VEL
LIN {X 0,Y 155.891,Z 293.098,A -85,B 0,C 180,E1 -28816.259,E2 -28816.259} C_VEL
LIN {X 0,Y 151.908,Z 306.115,A -85,B 0,C 180,E1 -28816.827,E2 -28816.827} C_VEL
LIN {X 0,Y 146.456,Z 318.868,A -85,B 0,C 180,E1 -28817.496,E2 -28817.496} C_VEL
LIN {X 0,Y 139.833,Z 330.86,A -85,B 0,C 180,E1 -28818.441,E2 -28818.441} C_VEL
LIN {X 0,Y 132.453,Z 341.49,A -85,B 0,C 180,E1 -28819.641,E2 -28819.641} C_VEL
LIN {X 0,Y 124.442,Z 351.067,A -85,B 0,C 180,E1 -28821.274,E2 -28821.274} C_VEL
LIN {X 0,Y 114.934,Z 360.43,A -85,B 0,C 180,E1 -28823.477,E2 -28823.477} C_VEL
LIN {X 0,Y 105.638,Z 367.944,A -85,B 0,C 180,E1 -28826.086,E2 -28826.086} C_VEL
LIN {X 0,Y 96.693,Z 374.03,A -85,B 0,C 180,E1 -28829.285,E2 -28829.285} C_VEL
LIN {X 0,Y 88.181,Z 378.912,A -85,B 0,C 180,E1 -28833.193,E2 -28833.193} C_VEL
LIN {X 0,Y 80.248,Z 382.73,A -85,B 0,C 180,E1 -28837.983,E2 -28837.983} C_VEL
LIN {X 0,Y 70.66,Z 386.326,A -85,B 0,C 180,E1 -28845.876,E2 -28845.876} C_VEL
LIN {X 0,Y 66.528,Z 387.53,A -85,B 0,C 180,E1 -28850.668,E2 -28850.668} C_VEL
LIN {X 0,Y 59.902,Z 388.741,A -85,B 0,C 180,E1 -28862.013,E2 -28862.013} C_VEL
LIN {X 0,Y 56.257,Z 388.489,A -85,B 0,C 180,E1 -28875.532,E2 -28875.532} C_VEL
LIN {X 0,Y 55.576,Z 387.779,A -85,B 0,C 180,E1 -28882.736,E2 -28882.736} C_VEL
LIN {X 0,Y 55.638,Z 386.65,A -85,B 0,C 180,E1 -28890.001,E2 -28890.001} C_VEL
LIN {X 0,Y 55.864,Z 384.101,A -85,B 0,C 180,E1 -28900.879,E2 -28900.879} C_VEL
LIN {X 0,Y 57.724,Z 380.5,A -85,B 0,C 180,E1 -28911.425,E2 -28911.425} C_VEL
LIN {X 0,Y 61.211,Z 375.749,A -85,B 0,C 180,E1 -28921.111,E2 -28921.111} C_VEL
LIN {X 0,Y 66.214,Z 369.717,A -85,B 0,C 180,E1 -28929.559,E2 -28929.559} C_VEL
LIN {X 0,Y 71.282,Z 363.448,A -85,B 0,C 180,E1 -28935.754,E2 -28935.754} C_VEL
LIN {X 0,Y 78.283,Z 354.477,A -85,B 0,C 180,E1 -28941.774,E2 -28941.774} C_VEL
LIN {X 0,Y 84.662,Z 345.093,A -85,B 0,C 180,E1 -28946.114,E2 -28946.114} C_VEL
LIN {X 0,Y 90.866,Z 334.691,A -85,B 0,C 180,E1 -28949.37,E2 -28949.37} C_VEL
LIN {X 0,Y 95.822,Z 324.708,A -85,B 0,C 180,E1 -28951.661,E2 -28951.661} C_VEL
LIN {X 0,Y 100.996,Z 312.122,A -85,B 0,C 180,E1 -28953.631,E2 -28953.631} C_VEL
LIN {X 0,Y 104.937,Z 298.967,A -85,B 0,C 180,E1 -28955.046,E2 -28955.046} C_VEL
LIN {X 0,Y 107.691,Z 285.271,A -85,B 0,C 180,E1 -28956.018,E2 -28956.018} C_VEL
LIN {X 0,Y 110.203,Z 262.289,A -85,B 0,C 180,E1 -28957.051,E2 -28957.051} C_VEL
LIN {X 0,Y 107.562,Z 252.528,A -85,B 0,C 180,E1 -28960.805,E2 -28960.805} C_VEL
LIN {X 0,Y 104.512,Z 245.743,A -85,B 0,C 180,E1 -28965.167,E2 -28965.167} C_VEL
LIN {X 0,Y 101.515,Z 239.835,A -85,B 0,C 180,E1 -28970.502,E2 -28970.502} C_VEL
LIN {X 0,Y 99.421,Z 235.832,A -85,B 0,C 180,E1 -28975.32,E2 -28975.32} C_VEL
LIN {X 0,Y 98.034,Z 232.708,A -85,B 0,C 180,E1 -28979.997,E2 -28979.997} C_VEL
LIN {X 0,Y 96.98,Z 231.423,A -85,B 0,C 180,E1 -28984.861,E2 -28984.861} C_VEL
LIN {X 0,Y 96.591,Z 230.925,A -85,B 0,C 180,E1 -28988.364,E2 -28988.364} C_VEL
LIN {X 0,Y 96.527,Z 231.385,A -85,B 0,C 180,E1 -28994.109,E2 -28994.109} C_VEL
LIN {X 0,Y 97.97,Z 233.27,A -85,B 0,C 180,E1 -29002.626,E2 -29002.626} C_VEL
LIN {X 0,Y 98.728,Z 236.018,A -85,B 0,C 180,E1 -29005.651,E2 -29005.651} C_VEL
LIN {X 0,Y 99.484,Z 239.576,A -85,B 0,C 180,E1 -29008.375,E2 -29008.375} C_VEL
LIN {X 0,Y 102.795,Z 253.058,A -85,B 0,C 180,E1 -29016.617,E2 -29016.617} C_VEL
LIN {X 0,Y 105.284,Z 259.038,A -85,B 0,C 180,E1 -29020.497,E2 -29020.497} C_VEL
LIN {X 0,Y 106.5,Z 262.23,A -85,B 0,C 180,E1 -29022.199,E2 -29022.199} C_VEL
LIN {X 0,Y 103.99,Z 282.745,A -85,B 0,C 180,E1 -29023.058,E2 -29023.058} C_VEL
LIN {X 0,Y 101.214,Z 295.885,A -85,B 0,C 180,E1 -29024.032,E2 -29024.032} C_VEL
LIN {X 0,Y 97.217,Z 308.898,A -85,B 0,C 180,E1 -29025.545,E2 -29025.545} C_VEL
LIN {X 0,Y 92.355,Z 320.74,A -85,B 0,C 180,E1 -29027.516,E2 -29027.516} C_VEL
LIN {X 0,Y 86.454,Z 332.219,A -85,B 0,C 180,E1 -29030.194,E2 -29030.194} C_VEL
LIN {X 0,Y 80.083,Z 342.447,A -85,B 0,C 180,E1 -29033.63,E2 -29033.63} C_VEL
LIN {X 0,Y 73.262,Z 351.807,A -85,B 0,C 180,E1 -29038.154,E2 -29038.154} C_VEL
LIN {X 0,Y 66.931,Z 359.476,A -85,B 0,C 180,E1 -29043.494,E2 -29043.494} C_VEL
LIN {X 0,Y 59.938,Z 367.28,A -85,B 0,C 180,E1 -29051.654,E2 -29051.654} C_VEL
LIN {X 0,Y 53.849,Z 373.807,A -85,B 0,C 180,E1 -29062.499,E2 -29062.499} C_VEL
LIN {X 0,Y 50.259,Z 378.038,A -85,B 0,C 180,E1 -29073.194,E2 -29073.194} C_VEL
LIN {X 0,Y 48.127,Z 381.679,A -85,B 0,C 180,E1 -29086.98,E2 -29086.98} C_VEL
LIN {X 0,Y 48.357,Z 383.812,A -85,B 0,C 180,E1 -29099.321,E2 -29099.321} C_VEL
LIN {X 0,Y 51.168,Z 385.24,A -85,B 0,C 180,E1 -29113.372,E2 -29113.372} C_VEL
LIN {X 0,Y 54.16,Z 385.526,A -85,B 0,C 180,E1 -29121.129,E2 -29121.129} C_VEL
LIN {X 0,Y 61.466,Z 384.838,A -85,B 0,C 180,E1 -29132.789,E2 -29132.789} C_VEL
LIN {X 0,Y 67.627,Z 383.536,A -85,B 0,C 180,E1 -29139.275,E2 -29139.275} C_VEL
LIN {X 0,Y 76.125,Z 380.908,A -85,B 0,C 180,E1 -29145.783,E2 -29145.783} C_VEL
LIN {X 0,Y 85.407,Z 377.095,A -85,B 0,C 180,E1 -29150.911,E2 -29150.911} C_VEL
LIN {X 0,Y 94.813,Z 372.223,A -85,B 0,C 180,E1 -29154.841,E2 -29154.841} C_VEL
LIN {X 0,Y 105.464,Z 365.385,A -85,B 0,C 180,E1 -29158.333,E2 -29158.333} C_VEL
LIN {X 0,Y 114.211,Z 358.525,A -85,B 0,C 180,E1 -29160.617,E2 -29160.617} C_VEL
LIN {X 0,Y 124.162,Z 348.991,A -85,B 0,C 180,E1 -29162.801,E2 -29162.801} C_VEL
LIN {X 0,Y 132.146,Z 339.692,A -85,B 0,C 180,E1 -29164.297,E2 -29164.297} C_VEL
LIN {X 0,Y 139.83,Z 328.722,A -85,B 0,C 180,E1 -29165.551,E2 -29165.551} C_VEL
LIN {X 0,Y 145.894,Z 317.849,A -85,B 0,C 180,E1 -29166.515,E2 -29166.515} C_VEL
LIN {X 0,Y 151.474,Z 304.97,A -85,B 0,C 180,E1 -29167.316,E2 -29167.316} C_VEL
LIN {X 0,Y 153.834,Z 297.953,A -85,B 0,C 180,E1 -29167.678,E2 -29167.678} C_VEL
LIN {X 0,Y 153.875,Z 297.113,A -85,B 0,C 180,E1 -29169.864,E2 -29169.864} C_VEL
LIN {X 0,Y 153.749,Z 297.648,A -85,B 0,C 180,E1 -29171.538,E2 -29171.538} C_VEL
LIN {X 0,Y 153.69,Z 298.464,A -85,B 0,C 180,E1 -29173.219,E2 -29173.219} C_VEL
LIN {X 0,Y 153.32,Z 300.015,A -85,B 0,C 180,E1 -29173.917,E2 -29173.917} C_VEL
LIN {X 0,Y 148.757,Z 312.16,A -85,B 0,C 180,E1 -29174.403,E2 -29174.403} C_VEL
LIN {X 0,Y 142.828,Z 324.164,A -85,B 0,C 180,E1 -29175.059,E2 -29175.059} C_VEL
LIN {X 0,Y 136.105,Z 334.964,A -85,B 0,C 180,E1 -29175.904,E2 -29175.904} C_VEL
LIN {X 0,Y 128.62,Z 344.749,A -85,B 0,C 180,E1 -29177.016,E2 -29177.016} C_VEL
LIN {X 0,Y 120.447,Z 353.666,A -85,B 0,C 180,E1 -29178.528,E2 -29178.528} C_VEL
LIN {X 0,Y 112.315,Z 361.114,A -85,B 0,C 180,E1 -29180.181,E2 -29180.181} C_VEL
LIN {X 0,Y 102.731,Z 368.464,A -85,B 0,C 180,E1 -29182.55,E2 -29182.55} C_VEL
LIN {X 0,Y 93.438,Z 374.403,A -85,B 0,C 180,E1 -29185.501,E2 -29185.501} C_VEL
LIN {X 0,Y 84.507,Z 379.144,A -85,B 0,C 180,E1 -29189.166,E2 -29189.166} C_VEL
LIN {X 0,Y 76.071,Z 382.827,A -85,B 0,C 180,E1 -29193.75,E2 -29193.75} C_VEL
LIN {X 0,Y 65.738,Z 386.292,A -85,B 0,C 180,E1 -29201.553,E2 -29201.553} C_VEL
LIN {X 0,Y 57.111,Z 388.137,A -85,B 0,C 180,E1 -29212.028,E2 -29212.028} C_VEL
LIN {X 0,Y 51.147,Z 388.512,A -85,B 0,C 180,E1 -29225.657,E2 -29225.657} C_VEL
LIN {X 0,Y 49.41,Z 388.13,A -85,B 0,C 180,E1 -29233.474,E2 -29233.474} C_VEL
LIN {X 0,Y 48.542,Z 387.339,A -85,B 0,C 180,E1 -29241.677,E2 -29241.677} C_VEL
LIN {X 0,Y 48.546,Z 386.162,A -85,B 0,C 180,E1 -29250.002,E2 -29250.002} C_VEL
LIN {X 0,Y 48.914,Z 383.509,A -85,B 0,C 180,E1 -29262.448,E2 -29262.448} C_VEL
LIN {X 0,Y 51.133,Z 379.794,A -85,B 0,C 180,E1 -29274.354,E2 -29274.354} C_VEL
LIN {X 0,Y 55.242,Z 374.93,A -85,B 0,C 180,E1 -29284.927,E2 -29284.927} C_VEL
LIN {X 0,Y 60.864,Z 368.764,A -85,B 0,C 180,E1 -29293.856,E2 -29293.856} C_VEL
LIN {X 0,Y 67.093,Z 361.621,A -85,B 0,C 180,E1 -29300.793,E2 -29300.793} C_VEL
LIN {X 0,Y 74.06,Z 353.18,A -85,B 0,C 180,E1 -29306.136,E2 -29306.136} C_VEL
LIN {X 0,Y 80.862,Z 343.507,A -85,B 0,C 180,E1 -29310.36,E2 -29310.36} C_VEL
LIN {X 0,Y 87.456,Z 332.86,A -85,B 0,C 180,E1 -29313.385,E2 -29313.385} C_VEL
LIN {X 0,Y 92.656,Z 322.527,A -85,B 0,C 180,E1 -29315.537,E2 -29315.537} C_VEL
LIN {X 0,Y 97.661,Z 310.292,A -85,B 0,C 180,E1 -29317.227,E2 -29317.227} C_VEL
LIN {X 0,Y 101.735,Z 296.603,A -85,B 0,C 180,E1 -29318.551,E2 -29318.551} C_VEL
LIN {X 0,Y 104.246,Z 283.457,A -85,B 0,C 180,E1 -29319.392,E2 -29319.392} C_VEL
LIN {X 0,Y 106.36,Z 264.52,A -85,B 0,C 180,E1 -29320.22,E2 -29320.22} C_VEL
LIN {X 0,Y 104.592,Z 257.391,A -85,B 0,C 180,E1 -29323.124,E2 -29323.124} C_VEL
LIN {X 0,Y 102.141,Z 251.423,A -85,B 0,C 180,E1 -29327.154,E2 -29327.154} C_VEL
LIN {X 0,Y 99.688,Z 246.13,A -85,B 0,C 180,E1 -29332.076,E2 -29332.076} C_VEL
LIN {X 0,Y 97.918,Z 242.355,A -85,B 0,C 180,E1 -29336.724,E2 -29336.724} C_VEL
LIN {X 0,Y 96.768,Z 239.467,A -85,B 0,C 180,E1 -29341.227,E2 -29341.227} C_VEL
LIN {X 0,Y 95.93,Z 238.359,A -85,B 0,C 180,E1 -29345.631,E2 -29345.631} C_VEL
LIN {X 0,Y 95.566,Z 238.019,A -85,B 0,C 180,E1 -29350.095,E2 -29350.095} C_VEL
LIN {X 0,Y 95.69,Z 238.748,A -85,B 0,C 180,E1 -29355.571,E2 -29355.571} C_VEL
LIN {X 0,Y 96.768,Z 240.238,A -85,B 0,C 180,E1 -29361.775,E2 -29361.775} C_VEL
LIN {X 0,Y 98.741,Z 244.431,A -85,B 0,C 180,E1 -29368.326,E2 -29368.326} C_VEL
LIN {X 0,Y 100.605,Z 248.298,A -85,B 0,C 180,E1 -29372.556,E2 -29372.556} C_VEL
LIN {X 0,Y 102.611,Z 252.635,A -85,B 0,C 180,E1 -29376.303,E2 -29376.303} C_VEL
LIN {X 0,Y 102.795,Z 253.058,A -85,B 0,C 180,E1 -29376.617,E2 -29376.617} C_VEL
LIN {X 0,Y 103.485,Z 255.916,A -85,B 0,C 180,E1 -29377.958,E2 -29377.958} C_VEL
LIN {X 0,Y 103.752,Z 259.42,A -85,B 0,C 180,E1 -29378.826,E2 -29378.826} C_VEL
LIN {X 0,Y 103.516,Z 265.249,A -85,B 0,C 180,E1 -29379.47,E2 -29379.47} C_VEL
LIN {X 0,Y 101.928,Z 275.801,A -85,B 0,C 180,E1 -29379.518,E2 -29379.518} C_VEL
LIN {X 0,Y 100.371,Z 284.333,A -85,B 0,C 180,E1 -29379.645,E2 -29379.645} C_VEL
LIN {X 0,Y 97.51,Z 296.985,A -85,B 0,C 180,E1 -29380.553,E2 -29380.553} C_VEL
LIN {X 0,Y 93.366,Z 309.713,A -85,B 0,C 180,E1 -29381.982,E2 -29381.982} C_VEL
LIN {X 0,Y 87.895,Z 322.266,A -85,B 0,C 180,E1 -29383.974,E2 -29383.974} C_VEL
LIN {X 0,Y 81.717,Z 333.466,A -85,B 0,C 180,E1 -29386.524,E2 -29386.524} C_VEL
LIN {X 0,Y 74.569,Z 344.174,A -85,B 0,C 180,E1 -29390.158,E2 -29390.158} C_VEL
LIN {X 0,Y 67.176,Z 353.564,A -85,B 0,C 180,E1 -29394.87,E2 -29394.87} C_VEL
LIN {X 0,Y 59.19,Z 362.278,A -85,B 0,C 180,E1 -29401.642,E2 -29401.642} C_VEL
LIN {X 0,Y 52.328,Z 369.103,A -85,B 0,C 180,E1 -29410.058,E2 -29410.058} C_VEL
LIN {X 0,Y 46.486,Z 374.834,A -85,B 0,C 180,E1 -29421.302,E2 -29421.302} C_VEL
LIN {X 0,Y 42.37,Z 379.406,A -85,B 0,C 180,E1 -29435.674,E2 -29435.674} C_VEL
LIN {X 0,Y 40.885,Z 382.38,A -85,B 0,C 180,E1 -29450.106,E2 -29450.106} C_VEL
LIN {X 0,Y 41.509,Z 384.081,A -85,B 0,C 180,E1 -29462.175,E2 -29462.175} C_VEL
LIN {X 0,Y 45.834,Z 385.627,A -85,B 0,C 180,E1 -29480.055,E2 -29480.055} C_VEL
LIN {X 0,Y 49.63,Z 385.772,A -85,B 0,C 180,E1 -29488.17,E2 -29488.17} C_VEL
LIN {X 0,Y 57.046,Z 385.122,A -85,B 0,C 180,E1 -29498.316,E2 -29498.316} C_VEL
LIN {X 0,Y 68.741,Z 382.559,A -85,B 0,C 180,E1 -29508.206,E2 -29508.206} C_VEL
LIN {X 0,Y 77.84,Z 379.516,A -85,B 0,C 180,E1 -29513.29,E2 -29513.29} C_VEL
LIN {X 0,Y 87.936,Z 375.096,A -85,B 0,C 180,E1 -29517.447,E2 -29517.447} C_VEL
LIN {X 0,Y 98.399,Z 369.31,A -85,B 0,C 180,E1 -29520.726,E2 -29520.726} C_VEL
LIN {X 0,Y 107.972,Z 362.801,A -85,B 0,C 180,E1 -29523.112,E2 -29523.112} C_VEL
LIN {X 0,Y 118.204,Z 354.263,A -85,B 0,C 180,E1 -29525.198,E2 -29525.198} C_VEL
LIN {X 0,Y 127.392,Z 344.813,A -85,B 0,C 180,E1 -29526.773,E2 -29526.773} C_VEL
LIN {X 0,Y 135.543,Z 334.556,A -85,B 0,C 180,E1 -29527.96,E2 -29527.96} C_VEL
LIN {X 0,Y 142.266,Z 324.055,A -85,B 0,C 180,E1 -29528.884,E2 -29528.884} C_VEL
LIN {X 0,Y 147.749,Z 313.369,A -85,B 0,C 180,E1 -29529.584,E2 -29529.584} C_VEL
LIN {X 0,Y 151.521,Z 304.216,A -85,B 0,C 180,E1 -29530.056,E2 -29530.056} C_VEL
LIN {X 0,Y 151.644,Z 303.853,A -85,B 0,C 180,E1 -29530.201,E2 -29530.201} C_VEL
LIN {X 0,Y 151.525,Z 304.254,A -85,B 0,C 180,E1 -29531.048,E2 -29531.048} C_VEL
LIN {X 0,Y 151.196,Z 305.189,A -85,B 0,C 180,E1 -29531.419,E2 -29531.419} C_VEL
LIN {X 0,Y 145.444,Z 318.312,A -85,B 0,C 180,E1 -29531.895,E2 -29531.895} C_VEL
LIN {X 0,Y 138.603,Z 330.295,A -85,B 0,C 180,E1 -29532.555,E2 -29532.555} C_VEL
LIN {X 0,Y 130.956,Z 340.908,A -85,B 0,C 180,E1 -29533.417,E2 -29533.417} C_VEL
LIN {X 0,Y 121.716,Z 351.358,A -85,B 0,C 180,E1 -29534.726,E2 -29534.726} C_VEL
LIN {X 0,Y 113.404,Z 359.112,A -85,B 0,C 180,E1 -29536.142,E2 -29536.142} C_VEL
LIN {X 0,Y 103.514,Z 366.778,A -85,B 0,C 180,E1 -29538.101,E2 -29538.101} C_VEL
LIN {X 0,Y 93.802,Z 372.974,A -85,B 0,C 180,E1 -29540.521,E2 -29540.521} C_VEL
LIN {X 0,Y 84.339,Z 377.962,A -85,B 0,C 180,E1 -29543.562,E2 -29543.562} C_VEL
LIN {X 0,Y 72.67,Z 382.833,A -85,B 0,C 180,E1 -29548.923,E2 -29548.923} C_VEL
LIN {X 0,Y 66.683,Z 384.804,A -85,B 0,C 180,E1 -29552.527,E2 -29552.527} C_VEL
LIN {X 0,Y 56.245,Z 387.279,A -85,B 0,C 180,E1 -29561.436,E2 -29561.436} C_VEL
LIN {X 0,Y 47.77,Z 388.272,A -85,B 0,C 180,E1 -29573.952,E2 -29573.952} C_VEL
LIN {X 0,Y 44.74,Z 388.205,A -85,B 0,C 180,E1 -29581.886,E2 -29581.886} C_VEL
LIN {X 0,Y 41.544,Z 386.896,A -85,B 0,C 180,E1 -29600.262,E2 -29600.262} C_VEL
LIN {X 0,Y 41.444,Z 385.664,A -85,B 0,C 180,E1 -29610.002,E2 -29610.002} C_VEL
LIN {X 0,Y 41.995,Z 382.899,A -85,B 0,C 180,E1 -29624.541,E2 -29624.541} C_VEL
LIN {X 0,Y 44.724,Z 379.062,A -85,B 0,C 180,E1 -29638.129,E2 -29638.129} C_VEL
LIN {X 0,Y 49.581,Z 374.076,A -85,B 0,C 180,E1 -29649.635,E2 -29649.635} C_VEL
LIN {X 0,Y 55.931,Z 367.766,A -85,B 0,C 180,E1 -29658.935,E2 -29658.935} C_VEL
LIN {X 0,Y 63.187,Z 360.083,A -85,B 0,C 180,E1 -29666.049,E2 -29666.049} C_VEL
LIN {X 0,Y 70.322,Z 351.741,A -85,B 0,C 180,E1 -29670.987,E2 -29670.987} C_VEL
LIN {X 0,Y 77.587,Z 341.842,A -85,B 0,C 180,E1 -29674.938,E2 -29674.938} C_VEL
LIN {X 0,Y 84.495,Z 330.846,A -85,B 0,C 180,E1 -29677.723,E2 -29677.723} C_VEL
LIN {X 0,Y 89.921,Z 320.017,A -85,B 0,C 180,E1 -29679.703,E2 -29679.703} C_VEL
LIN {X 0,Y 95.121,Z 307.106,A -85,B 0,C 180,E1 -29681.203,E2 -29681.203} C_VEL
LIN {X 0,Y 98.769,Z 294.375,A -85,B 0,C 180,E1 -29682.254,E2 -29682.254} C_VEL
LIN {X 0,Y 101.217,Z 280.844,A -85,B 0,C 180,E1 -29682.987,E2 -29682.987} C_VEL
LIN {X 0,Y 102.834,Z 266.868,A -85,B 0,C 180,E1 -29683.534,E2 -29683.534} C_VEL
LIN {X 0,Y 101.64,Z 261.707,A -85,B 0,C 180,E1 -29685.876,E2 -29685.876} C_VEL
LIN {X 0,Y 99.359,Z 255.688,A -85,B 0,C 180,E1 -29690.406,E2 -29690.406} C_VEL
LIN {X 0,Y 97.453,Z 251.411,A -85,B 0,C 180,E1 -29694.982,E2 -29694.982} C_VEL
LIN {X 0,Y 96.401,Z 248.727,A -85,B 0,C 180,E1 -29698.439,E2 -29698.439} C_VEL
LIN {X 0,Y 95.586,Z 246.3,A -85,B 0,C 180,E1 -29702.209,E2 -29702.209} C_VEL
LIN {X 0,Y 94.824,Z 245.182,A -85,B 0,C 180,E1 -29707.15,E2 -29707.15} C_VEL
LIN {X 0,Y 94.628,Z 245.294,A -85,B 0,C 180,E1 -29712.87,E2 -29712.87} C_VEL
LIN {X 0,Y 95.577,Z 247.138,A -85,B 0,C 180,E1 -29720.826,E2 -29720.826} C_VEL
LIN {X 0,Y 97.248,Z 251.084,A -85,B 0,C 180,E1 -29727.08,E2 -29727.08} C_VEL
LIN {X 0,Y 99.411,Z 255.97,A -85,B 0,C 180,E1 -29732.37,E2 -29732.37} C_VEL
LIN {X 0,Y 101.869,Z 262.336,A -85,B 0,C 180,E1 -29737.136,E2 -29737.136} C_VEL
LIN {X 0,Y 102.887,Z 265.187,A -85,B 0,C 180,E1 -29738.859,E2 -29738.859} C_VEL
LIN {X 0,Y 100.551,Z 283.354,A -85,B 0,C 180,E1 -29739.6,E2 -29739.6} C_VEL
LIN {X 0,Y 100.371,Z 284.333,A -85,B 0,C 180,E1 -29739.645,E2 -29739.645} C_VEL
LIN {X 0,Y 98.946,Z 290.066,A -85,B 0,C 180,E1 -29739.668,E2 -29739.668} C_VEL
LIN {X 0,Y 95.292,Z 299.194,A -85,B 0,C 180,E1 -29738.865,E2 -29738.865} C_VEL
LIN {X 0,Y 91.089,Z 308.129,A -85,B 0,C 180,E1 -29738.163,E2 -29738.163} C_VEL
LIN {X 0,Y 88.712,Z 313.518,A -85,B 0,C 180,E1 -29738.522,E2 -29738.522} C_VEL
LIN {X 0,Y 83.005,Z 325.229,A -85,B 0,C 180,E1 -29740.355,E2 -29740.355} C_VEL
LIN {X 0,Y 75.826,Z 337.072,A -85,B 0,C 180,E1 -29743.12,E2 -29743.12} C_VEL
LIN {X 0,Y 68.367,Z 347.129,A -85,B 0,C 180,E1 -29746.665,E2 -29746.665} C_VEL
LIN {X 0,Y 59.861,Z 356.773,A -85,B 0,C 180,E1 -29751.946,E2 -29751.946} C_VEL
LIN {X 0,Y 52.815,Z 363.69,A -85,B 0,C 180,E1 -29757.839,E2 -29757.839} C_VEL
LIN {X 0,Y 46.262,Z 369.587,A -85,B 0,C 180,E1 -29765.697,E2 -29765.697} C_VEL
LIN {X 0,Y 41.01,Z 374.145,A -85,B 0,C 180,E1 -29775.102,E2 -29775.102} C_VEL
LIN {X 0,Y 36.127,Z 378.689,A -85,B 0,C 180,E1 -29789.998,E2 -29789.998} C_VEL
LIN {X 0,Y 34.255,Z 381.11,A -85,B 0,C 180,E1 -29801.837,E2 -29801.837} C_VEL
LIN {X 0,Y 33.816,Z 383.002,A -85,B 0,C 180,E1 -29814.559,E2 -29814.559} C_VEL
LIN {X 0,Y 34.933,Z 384.44,A -85,B 0,C 180,E1 -29827.123,E2 -29827.123} C_VEL
LIN {X 0,Y 37.49,Z 385.446,A -85,B 0,C 180,E1 -29838.574,E2 -29838.574} C_VEL
LIN {X 0,Y 41.98,Z 385.991,A -85,B 0,C 180,E1 -29849.861,E2 -29849.861} C_VEL
LIN {X 0,Y 51.443,Z 385.648,A -85,B 0,C 180,E1 -29862.999,E2 -29862.999} C_VEL
LIN {X 0,Y 57.415,Z 384.764,A -85,B 0,C 180,E1 -29868.304,E2 -29868.304} C_VEL
LIN {X 0,Y 65.955,Z 382.88,A -85,B 0,C 180,E1 -29873.888,E2 -29873.888} C_VEL
LIN {X 0,Y 77.317,Z 379.235,A -85,B 0,C 180,E1 -29879.061,E2 -29879.061} C_VEL
LIN {X 0,Y 87.935,Z 374.663,A -85,B 0,C 180,E1 -29882.53,E2 -29882.53} C_VEL
LIN {X 0,Y 98.804,Z 368.708,A -85,B 0,C 180,E1 -29885.242,E2 -29885.242} C_VEL
LIN {X 0,Y 109.602,Z 361.243,A -85,B 0,C 180,E1 -29887.371,E2 -29887.371} C_VEL
LIN {X 0,Y 119.153,Z 353.13,A -85,B 0,C 180,E1 -29888.9,E2 -29888.9} C_VEL
LIN {X 0,Y 128.529,Z 343.399,A -85,B 0,C 180,E1 -29890.185,E2 -29890.185} C_VEL
LIN {X 0,Y 128.649,Z 343.279,A -85,B 0,C 180,E1 -29890.48,E2 -29890.48} C_VEL
LIN {X 0,Y 120.126,Z 352.36,A -85,B 0,C 180,E1 -29891.491,E2 -29891.491} C_VEL
LIN {X 0,Y 109.953,Z 361.245,A -85,B 0,C 180,E1 -29892.905,E2 -29892.905} C_VEL
LIN {X 0,Y 99.871,Z 368.457,A -85,B 0,C 180,E1 -29894.627,E2 -29894.627} C_VEL
LIN {X 0,Y 88.264,Z 375.142,A -85,B 0,C 180,E1 -29897.16,E2 -29897.16} C_VEL
LIN {X 0,Y 78.566,Z 379.606,A -85,B 0,C 180,E1 -29900.075,E2 -29900.075} C_VEL
LIN {X 0,Y 68.476,Z 383.264,A -85,B 0,C 180,E1 -29904.244,E2 -29904.244} C_VEL
LIN {X 0,Y 57.301,Z 386.168,A -85,B 0,C 180,E1 -29910.847,E2 -29910.847} C_VEL
LIN {X 0,Y 46.716,Z 387.782,A -85,B 0,C 180,E1 -29921.22,E2 -29921.22} C_VEL
LIN {X 0,Y 42.213,Z 388.015,A -85,B 0,C 180,E1 -29928.246,E2 -29928.246} C_VEL
LIN {X 0,Y 35.978,Z 387.341,A -85,B 0,C 180,E1 -29947.005,E2 -29947.005} C_VEL
LIN {X 0,Y 34.564,Z 386.45,A -85,B 0,C 180,E1 -29958.27,E2 -29958.27} C_VEL
LIN {X 0,Y 34.361,Z 385.166,A -85,B 0,C 180,E1 -29970.002,E2 -29970.002} C_VEL
LIN {X 0,Y 35.167,Z 382.29,A -85,B 0,C 180,E1 -29987.446,E2 -29987.446} C_VEL
LIN {X 0,Y 38.584,Z 378.333,A -85,B 0,C 180,E1 -30003.126,E2 -30003.126} C_VEL
LIN {X 0,Y 45.457,Z 372.216,A -85,B 0,C 180,E1 -30017.258,E2 -30017.258} C_VEL
LIN {X 0,Y 52.855,Z 365.477,A -85,B 0,C 180,E1 -30026.21,E2 -30026.21} C_VEL
LIN {X 0,Y 59.872,Z 358.468,A -85,B 0,C 180,E1 -30031.99,E2 -30031.99} C_VEL
LIN {X 0,Y 67.155,Z 350.308,A -85,B 0,C 180,E1 -30036.311,E2 -30036.311} C_VEL
LIN {X 0,Y 74.852,Z 340.154,A -85,B 0,C 180,E1 -30039.875,E2 -30039.875} C_VEL
LIN {X 0,Y 81.242,Z 330.133,A -85,B 0,C 180,E1 -30042.1,E2 -30042.1} C_VEL
LIN {X 0,Y 86.892,Z 319.215,A -85,B 0,C 180,E1 -30043.842,E2 -30043.842} C_VEL
LIN {X 0,Y 91.839,Z 307.278,A -85,B 0,C 180,E1 -30045.049,E2 -30045.049} C_VEL
LIN {X 0,Y 95.725,Z 294.188,A -85,B 0,C 180,E1 -30046.037,E2 -30046.037} C_VEL
LIN {X 0,Y 98.179,Z 281.288,A -85,B 0,C 180,E1 -30046.66,E2 -30046.66} C_VEL
LIN {X 0,Y 99.598,Z 269.072,A -85,B 0,C 180,E1 -30047.196,E2 -30047.196} C_VEL
LIN {X 0,Y 99.051,Z 266.621,A -85,B 0,C 180,E1 -30048.486,E2 -30048.486} C_VEL
LIN {X 0,Y 97.324,Z 261.488,A -85,B 0,C 180,E1 -30052.5,E2 -30052.5} C_VEL
LIN {X 0,Y 95.63,Z 257.046,A -85,B 0,C 180,E1 -30057.483,E2 -30057.483} C_VEL
LIN {X 0,Y 94.901,Z 254.843,A -85,B 0,C 180,E1 -30060.573,E2 -30060.573} C_VEL
LIN {X 0,Y 94.384,Z 253.035,A -85,B 0,C 180,E1 -30063.497,E2 -30063.497} C_VEL
LIN {X 0,Y 93.788,Z 252.041,A -85,B 0,C 180,E1 -30068.616,E2 -30068.616} C_VEL
LIN {X 0,Y 93.762,Z 252.77,A -85,B 0,C 180,E1 -30074.811,E2 -30074.811} C_VEL
LIN {X 0,Y 94.399,Z 253.956,A -85,B 0,C 180,E1 -30079.753,E2 -30079.753} C_VEL
LIN {X 0,Y 95.73,Z 257.523,A -85,B 0,C 180,E1 -30085.538,E2 -30085.538} C_VEL
LIN {X 0,Y 97.469,Z 262.026,A -85,B 0,C 180,E1 -30090.521,E2 -30090.521} C_VEL
LIN {X 0,Y 99.527,Z 268.029,A -85,B 0,C 180,E1 -30095.094,E2 -30095.094} C_VEL
LIN {X 0,Y 99.635,Z 268.357,A -85,B 0,C 180,E1 -30095.314,E2 -30095.314} C_VEL
LIN {X 0,Y 97.196,Z 285.568,A -85,B 0,C 180,E1 -30095.973,E2 -30095.973} C_VEL
LIN {X 0,Y 94.123,Z 298.277,A -85,B 0,C 180,E1 -30096.841,E2 -30096.841} C_VEL
LIN {X 0,Y 89.496,Z 311.54,A -85,B 0,C 180,E1 -30098.251,E2 -30098.251} C_VEL
LIN {X 0,Y 88.712,Z 313.518,A -85,B 0,C 180,E1 -30098.522,E2 -30098.522} C_VEL
LIN {X 0,Y 86.144,Z 318.814,A -85,B 0,C 180,E1 -30098.884,E2 -30098.884} C_VEL
LIN {X 0,Y 80.611,Z 327.045,A -85,B 0,C 180,E1 -30098.432,E2 -30098.432} C_VEL
LIN {X 0,Y 74.438,Z 334.848,A -85,B 0,C 180,E1 -30098.101,E2 -30098.101} C_VEL
LIN {X 0,Y 70.858,Z 339.477,A -85,B 0,C 180,E1 -30098.84,E2 -30098.84} C_VEL
LIN {X 0,Y 62.376,Z 349.961,A -85,B 0,C 180,E1 -30102.527,E2 -30102.527} C_VEL
LIN {X 0,Y 54.244,Z 358.329,A -85,B 0,C 180,E1 -30107.138,E2 -30107.138} C_VEL
LIN {X 0,Y 45.345,Z 366.179,A -85,B 0,C 180,E1 -30114.461,E2 -30114.461} C_VEL
LIN {X 0,Y 37.468,Z 372.389,A -85,B 0,C 180,E1 -30124.737,E2 -30124.737} C_VEL
LIN {X 0,Y 31.817,Z 376.714,A -85,B 0,C 180,E1 -30137.236,E2 -30137.236} C_VEL
LIN {X 0,Y 28.138,Z 380.001,A -85,B 0,C 180,E1 -30152.748,E2 -30152.748} C_VEL
LIN {X 0,Y 27.038,Z 383.613,A -85,B 0,C 180,E1 -30181.32,E2 -30181.32} C_VEL
LIN {X 0,Y 29.154,Z 384.98,A -85,B 0,C 180,E1 -30196.315,E2 -30196.315} C_VEL
LIN {X 0,Y 32.863,Z 385.849,A -85,B 0,C 180,E1 -30208.803,E2 -30208.803} C_VEL
LIN {X 0,Y 37.761,Z 386.273,A -85,B 0,C 180,E1 -30218.52,E2 -30218.52} C_VEL
LIN {X 0,Y 43.466,Z 386.266,A -85,B 0,C 180,E1 -30225.957,E2 -30225.957} C_VEL
LIN {X 0,Y 50.045,Z 385.717,A -85,B 0,C 180,E1 -30231.934,E2 -30231.934} C_VEL
LIN {X 0,Y 56.349,Z 384.796,A -85,B 0,C 180,E1 -30236.169,E2 -30236.169} C_VEL
LIN {X 0,Y 63.873,Z 383.223,A -85,B 0,C 180,E1 -30240.005,E2 -30240.005} C_VEL
LIN {X 0,Y 73.952,Z 380.28,A -85,B 0,C 180,E1 -30243.758,E2 -30243.758} C_VEL
LIN {X 0,Y 84.923,Z 375.948,A -85,B 0,C 180,E1 -30246.749,E2 -30246.749} C_VEL
LIN {X 0,Y 96.404,Z 370.064,A -85,B 0,C 180,E1 -30249.103,E2 -30249.103} C_VEL
LIN {X 0,Y 99.82,Z 368.027,A -85,B 0,C 180,E1 -30249.705,E2 -30249.705} C_VEL
LIN {X 0,Y 100.027,Z 367.929,A -85,B 0,C 180,E1 -30250.377,E2 -30250.377} C_VEL
LIN {X 0,Y 89.819,Z 373.808,A -85,B 0,C 180,E1 -30252.023,E2 -30252.023} C_VEL
LIN {X 0,Y 79.735,Z 378.494,A -85,B 0,C 180,E1 -30254.175,E2 -30254.175} C_VEL
LIN {X 0,Y 69.869,Z 382.124,A -85,B 0,C 180,E1 -30257.144,E2 -30257.144} C_VEL
LIN {X 0,Y 60.228,Z 384.81,A -85,B 0,C 180,E1 -30261.013,E2 -30261.013} C_VEL
LIN {X 0,Y 48.008,Z 387.041,A -85,B 0,C 180,E1 -30268.558,E2 -30268.558} C_VEL
LIN {X 0,Y 37.198,Z 387.725,A -85,B 0,C 180,E1 -30280.913,E2 -30280.913} C_VEL
LIN {X 0,Y 29.562,Z 386.94,A -85,B 0,C 180,E1 -30301.613,E2 -30301.613} C_VEL
LIN {X 0,Y 27.637,Z 385.991,A -85,B 0,C 180,E1 -30315.271,E2 -30315.271} C_VEL
LIN {X 0,Y 27.26,Z 384.61,A -85,B 0,C 180,E1 -30330.003,E2 -30330.003} C_VEL
LIN {X 0,Y 28.449,Z 381.631,A -85,B 0,C 180,E1 -30351.753,E2 -30351.753} C_VEL
LIN {X 0,Y 32.848,Z 377.549,A -85,B 0,C 180,E1 -30369.934,E2 -30369.934} C_VEL
LIN {X 0,Y 40.948,Z 371.262,A -85,B 0,C 180,E1 -30384.617,E2 -30384.617} C_VEL
LIN {X 0,Y 49.232,Z 364.369,A -85,B 0,C 180,E1 -30393.156,E2 -30393.156} C_VEL
LIN {X 0,Y 56.252,Z 357.803,A -85,B 0,C 180,E1 -30397.981,E2 -30397.981} C_VEL
LIN {X 0,Y 64.612,Z 348.825,A -85,B 0,C 180,E1 -30402.137,E2 -30402.137} C_VEL
LIN {X 0,Y 72.718,Z 338.32,A -85,B 0,C 180,E1 -30405.127,E2 -30405.127} C_VEL
LIN {X 0,Y 79.331,Z 327.942,A -85,B 0,C 180,E1 -30407.038,E2 -30407.038} C_VEL
LIN {X 0,Y 85.191,Z 316.607,A -85,B 0,C 180,E1 -30408.428,E2 -30408.428} C_VEL
LIN {X 0,Y 90.026,Z 304.459,A -85,B 0,C 180,E1 -30409.403,E2 -30409.403} C_VEL
LIN {X 0,Y 93.803,Z 291.066,A -85,B 0,C 180,E1 -30410.169,E2 -30410.169} C_VEL
LIN {X 0,Y 96.016,Z 278.397,A -85,B 0,C 180,E1 -30410.674,E2 -30410.674} C_VEL
LIN {X 0,Y 96.787,Z 271.955,A -85,B 0,C 180,E1 -30410.891,E2 -30410.891} C_VEL
LIN {X 0,Y 95.45,Z 267.388,A -85,B 0,C 180,E1 -30414.595,E2 -30414.595} C_VEL
LIN {X 0,Y 93.966,Z 262.45,A -85,B 0,C 180,E1 -30420.287,E2 -30420.287} C_VEL
LIN {X 0,Y 93.206,Z 259.639,A -85,B 0,C 180,E1 -30425.058,E2 -30425.058} C_VEL
LIN {X 0,Y 92.789,Z 259.101,A -85,B 0,C 180,E1 -30430.047,E2 -30430.047} C_VEL
LIN {X 0,Y 93.228,Z 260.545,A -85,B 0,C 180,E1 -30438.355,E2 -30438.355} C_VEL
LIN {X 0,Y 94.313,Z 264.066,A -85,B 0,C 180,E1 -30444.076,E2 -30444.076} C_VEL
LIN {X 0,Y 95.716,Z 268.379,A -85,B 0,C 180,E1 -30448.853,E2 -30448.853} C_VEL
LIN {X 0,Y 96.705,Z 271.607,A -85,B 0,C 180,E1 -30451.515,E2 -30451.515} C_VEL
LIN {X 0,Y 94.411,Z 286.668,A -85,B 0,C 180,E1 -30452.058,E2 -30452.058} C_VEL
LIN {X 0,Y 91.438,Z 298.444,A -85,B 0,C 180,E1 -30452.787,E2 -30452.787} C_VEL
LIN {X 0,Y 86.865,Z 311.232,A -85,B 0,C 180,E1 -30453.969,E2 -30453.969} C_VEL
LIN {X 0,Y 80.994,Z 323.583,A -85,B 0,C 180,E1 -30455.559,E2 -30455.559} C_VEL
LIN {X 0,Y 74.334,Z 334.566,A -85,B 0,C 180,E1 -30457.642,E2 -30457.642} C_VEL
LIN {X 0,Y 70.858,Z 339.477,A -85,B 0,C 180,E1 -30458.84,E2 -30458.84} C_VEL
LIN {X 0,Y 67.148,Z 343.992,A -85,B 0,C 180,E1 -30459.753,E2 -30459.753} C_VEL
LIN {X 0,Y 59.99,Z 350.861,A -85,B 0,C 180,E1 -30460.029,E2 -30460.029} C_VEL
LIN {X 0,Y 52.333,Z 357.2,A -85,B 0,C 180,E1 -30460.455,E2 -30460.455} C_VEL
LIN {X 0,Y 47.883,Z 360.838,A -85,B 0,C 180,E1 -30461.987,E2 -30461.987} C_VEL
LIN {X 0,Y 39.677,Z 367.358,A -85,B 0,C 180,E1 -30468.168,E2 -30468.168} C_VEL
LIN {X 0,Y 32.192,Z 372.598,A -85,B 0,C 180,E1 -30476.918,E2 -30476.918} C_VEL
LIN {X 0,Y 24.575,Z 377.624,A -85,B 0,C 180,E1 -30493.379,E2 -30493.379} C_VEL
LIN {X 0,Y 19.988,Z 381.475,A -85,B 0,C 180,E1 -30520.121,E2 -30520.121} C_VEL
LIN {X 0,Y 22.271,Z 384.831,A -85,B 0,C 180,E1 -30560.885,E2 -30560.885} C_VEL
LIN {X 0,Y 29.587,Z 386.24,A -85,B 0,C 180,E1 -30581.825,E2 -30581.825} C_VEL
LIN {X 0,Y 35.652,Z 386.593,A -85,B 0,C 180,E1 -30590.268,E2 -30590.268} C_VEL
LIN {X 0,Y 47.833,Z 386.02,A -85,B 0,C 180,E1 -30600.007,E2 -30600.007} C_VEL
LIN {X 0,Y 56.373,Z 384.834,A -85,B 0,C 180,E1 -30604.189,E2 -30604.189} C_VEL
LIN {X 0,Y 67.403,Z 382.345,A -85,B 0,C 180,E1 -30607.888,E2 -30607.888} C_VEL
LIN {X 0,Y 73.495,Z 380.5,A -85,B 0,C 180,E1 -30609.426,E2 -30609.426} C_VEL
LIN {X 0,Y 71.491,Z 381.194,A -85,B 0,C 180,E1 -30610.565,E2 -30610.565} C_VEL
LIN {X 0,Y 58.056,Z 384.823,A -85,B 0,C 180,E1 -30614.436,E2 -30614.436} C_VEL
LIN {X 0,Y 51.479,Z 386.062,A -85,B 0,C 180,E1 -30617.132,E2 -30617.132} C_VEL
LIN {X 0,Y 38.834,Z 387.346,A -85,B 0,C 180,E1 -30625.197,E2 -30625.197} C_VEL
LIN {X 0,Y 27.785,Z 387.17,A -85,B 0,C 180,E1 -30640.643,E2 -30640.643} C_VEL
LIN {X 0,Y 23.556,Z 386.539,A -85,B 0,C 180,E1 -30653.369,E2 -30653.369} C_VEL
LIN {X 0,Y 20.849,Z 385.494,A -85,B 0,C 180,E1 -30670.304,E2 -30670.304} C_VEL
LIN {X 0,Y 20.174,Z 384.037,A -85,B 0,C 180,E1 -30690.004,E2 -30690.004} C_VEL
LIN {X 0,Y 22,Z 380.933,A -85,B 0,C 180,E1 -30718.637,E2 -30718.637} C_VEL
LIN {X 0,Y 27.754,Z 376.717,A -85,B 0,C 180,E1 -30739.44,E2 -30739.44} C_VEL
LIN {X 0,Y 37.27,Z 370.288,A -85,B 0,C 180,E1 -30753.605,E2 -30753.605} C_VEL
LIN {X 0,Y 46.43,Z 363.201,A -85,B 0,C 180,E1 -30761.101,E2 -30761.101} C_VEL
LIN {X 0,Y 56.151,Z 354.337,A -85,B 0,C 180,E1 -30765.933,E2 -30765.933} C_VEL
LIN {X 0,Y 65.302,Z 344.232,A -85,B 0,C 180,E1 -30769.14,E2 -30769.14} C_VEL
LIN {X 0,Y 72.934,Z 333.939,A -85,B 0,C 180,E1 -30771.012,E2 -30771.012} C_VEL
LIN {X 0,Y 79.76,Z 322.506,A -85,B 0,C 180,E1 -30772.44,E2 -30772.44} C_VEL
LIN {X 0,Y 85.528,Z 310.252,A -85,B 0,C 180,E1 -30773.358,E2 -30773.358} C_VEL
LIN {X 0,Y 90.135,Z 296.697,A -85,B 0,C 180,E1 -30774.088,E2 -30774.088} C_VEL
LIN {X 0,Y 93.157,Z 283.304,A -85,B 0,C 180,E1 -30774.58,E2 -30774.58} C_VEL
LIN {X 0,Y 94.219,Z 275.241,A -85,B 0,C 180,E1 -30774.936,E2 -30774.936} C_VEL
LIN {X 0,Y 93.038,Z 270.742,A -85,B 0,C 180,E1 -30779.674,E2 -30779.674} C_VEL
LIN {X 0,Y 92.406,Z 268.001,A -85,B 0,C 180,E1 -30783.446,E2 -30783.446} C_VEL
LIN {X 0,Y 92.163,Z 266.569,A -85,B 0,C 180,E1 -30785.862,E2 -30785.862} C_VEL
LIN {X 0,Y 91.857,Z 266.15,A -85,B 0,C 180,E1 -30790.15,E2 -30790.15} C_VEL
LIN {X 0,Y 92.173,Z 267.686,A -85,B 0,C 180,E1 -30797.754,E2 -30797.754} C_VEL
LIN {X 0,Y 92.973,Z 270.714,A -85,B 0,C 180,E1 -30802.712,E2 -30802.712} C_VEL
LIN {X 0,Y 94.128,Z 275.035,A -85,B 0,C 180,E1 -30807.405,E2 -30807.405} C_VEL
LIN {X 0,Y 94.18,Z 275.34,A -85,B 0,C 180,E1 -30807.614,E2 -30807.614} C_VEL
LIN {X 0,Y 91.823,Z 288.707,A -85,B 0,C 180,E1 -30807.983,E2 -30807.983} C_VEL
LIN {X 0,Y 88.159,Z 301.81,A -85,B 0,C 180,E1 -30808.724,E2 -30808.724} C_VEL
LIN {X 0,Y 83.906,Z 312.861,A -85,B 0,C 180,E1 -30809.65,E2 -30809.65} C_VEL
LIN {X 0,Y 77.835,Z 324.882,A -85,B 0,C 180,E1 -30810.928,E2 -30810.928} C_VEL
LIN {X 0,Y 70.976,Z 335.656,A -85,B 0,C 180,E1 -30812.681,E2 -30812.681} C_VEL
LIN {X 0,Y 63.316,Z 345.513,A -85,B 0,C 180,E1 -30815.051,E2 -30815.051} C_VEL
LIN {X 0,Y 55.623,Z 353.781,A -85,B 0,C 180,E1 -30818.069,E2 -30818.069} C_VEL
LIN {X 0,Y 47.883,Z 360.838,A -85,B 0,C 180,E1 -30821.987,E2 -30821.987} C_VEL
LIN {X 0,Y 43.343,Z 364.314,A -85,B 0,C 180,E1 -30823.916,E2 -30823.916} C_VEL
LIN {X 0,Y 34.933,Z 369.402,A -85,B 0,C 180,E1 -30825.968,E2 -30825.968} C_VEL
LIN {X 0,Y 26.234,Z 373.863,A -85,B 0,C 180,E1 -30829.641,E2 -30829.641} C_VEL
LIN {X 0,Y 21.463,Z 376.288,A -85,B 0,C 180,E1 -30835.79,E2 -30835.79} C_VEL
LIN {X 0,Y 14.138,Z 380.534,A -85,B 0,C 180,E1 -30863.619,E2 -30863.619} C_VEL
LIN {X 0,Y 12.725,Z 383.159,A -85,B 0,C 180,E1 -30903.517,E2 -30903.517} C_VEL
LIN {X 0,Y 17.17,Z 385.067,A -85,B 0,C 180,E1 -30935.859,E2 -30935.859} C_VEL
LIN {X 0,Y 28.147,Z 386.63,A -85,B 0,C 180,E1 -30957.09,E2 -30957.09} C_VEL
LIN {X 0,Y 35.186,Z 386.872,A -85,B 0,C 180,E1 -30962.965,E2 -30962.965} C_VEL
LIN {X 0,Y 46.666,Z 386.322,A -85,B 0,C 180,E1 -30968.669,E2 -30968.669} C_VEL
LIN {X 0,Y 43.053,Z 386.724,A -85,B 0,C 180,E1 -30971.644,E2 -30971.644} C_VEL
LIN {X 0,Y 29.872,Z 387.145,A -85,B 0,C 180,E1 -30979.773,E2 -30979.773} C_VEL
LIN {X 0,Y 23.765,Z 386.816,A -85,B 0,C 180,E1 -30987.484,E2 -30987.484} C_VEL
LIN {X 0,Y 14.374,Z 384.969,A -85,B 0,C 180,E1 -31020.736,E2 -31020.736} C_VEL
LIN {X 0,Y 13.082,Z 383.456,A -85,B 0,C 180,E1 -31050.006,E2 -31050.006} C_VEL
LIN {X 0,Y 16.126,Z 380.229,A -85,B 0,C 180,E1 -31090.83,E2 -31090.83} C_VEL
LIN {X 0,Y 23.745,Z 375.882,A -85,B 0,C 180,E1 -31112.623,E2 -31112.623} C_VEL
LIN {X 0,Y 33.07,Z 370.331,A -85,B 0,C 180,E1 -31123.014,E2 -31123.014} C_VEL
LIN {X 0,Y 42.95,Z 363.34,A -85,B 0,C 180,E1 -31129.059,E2 -31129.059} C_VEL
LIN {X 0,Y 52.026,Z 355.643,A -85,B 0,C 180,E1 -31132.36,E2 -31132.36} C_VEL
LIN {X 0,Y 61.748,Z 345.567,A -85,B 0,C 180,E1 -31134.828,E2 -31134.828} C_VEL
LIN {X 0,Y 69.553,Z 335.684,A -85,B 0,C 180,E1 -31136.241,E2 -31136.241} C_VEL
LIN {X 0,Y 76.518,Z 324.753,A -85,B 0,C 180,E1 -31137.275,E2 -31137.275} C_VEL
LIN {X 0,Y 82.635,Z 312.583,A -85,B 0,C 180,E1 -31137.929,E2 -31137.929} C_VEL
LIN {X 0,Y 87.188,Z 300.63,A -85,B 0,C 180,E1 -31138.381,E2 -31138.381} C_VEL
LIN {X 0,Y 90.584,Z 287.862,A -85,B 0,C 180,E1 -31138.76,E2 -31138.76} C_VEL
LIN {X 0,Y 91.995,Z 279.806,A -85,B 0,C 180,E1 -31138.985,E2 -31138.985} C_VEL
LIN {X 0,Y 92.041,Z 278.922,A -85,B 0,C 180,E1 -31139.279,E2 -31139.279} C_VEL
LIN {X 0,Y 91.272,Z 274.702,A -85,B 0,C 180,E1 -31144.702,E2 -31144.702} C_VEL
LIN {X 0,Y 91.105,Z 273.439,A -85,B 0,C 180,E1 -31147.038,E2 -31147.038} C_VEL
LIN {X 0,Y 90.924,Z 273.214,A -85,B 0,C 180,E1 -31150.256,E2 -31150.256} C_VEL
LIN {X 0,Y 91.11,Z 274.549,A -85,B 0,C 180,E1 -31156.767,E2 -31156.767} C_VEL
LIN {X 0,Y 91.683,Z 277.433,A -85,B 0,C 180,E1 -31161.445,E2 -31161.445} C_VEL
LIN {X 0,Y 91.994,Z 279.038,A -85,B 0,C 180,E1 -31163.317,E2 -31163.317} C_VEL
LIN {X 0,Y 89.576,Z 291.304,A -85,B 0,C 180,E1 -31163.739,E2 -31163.739} C_VEL
LIN {X 0,Y 85.989,Z 303.282,A -85,B 0,C 180,E1 -31164.287,E2 -31164.287} C_VEL
LIN {X 0,Y 81.428,Z 314.481,A -85,B 0,C 180,E1 -31164.999,E2 -31164.999} C_VEL
LIN {X 0,Y 75.234,Z 326.133,A -85,B 0,C 180,E1 -31165.953,E2 -31165.953} C_VEL
LIN {X 0,Y 67.283,Z 337.959,A -85,B 0,C 180,E1 -31167.391,E2 -31167.391} C_VEL
LIN {X 0,Y 58.535,Z 348.341,A -85,B 0,C 180,E1 -31169.482,E2 -31169.482} C_VEL
LIN {X 0,Y 49.818,Z 356.824,A -85,B 0,C 180,E1 -31172.17,E2 -31172.17} C_VEL
LIN {X 0,Y 39.514,Z 365.126,A -85,B 0,C 180,E1 -31176.831,E2 -31176.831} C_VEL
LIN {X 0,Y 29.488,Z 371.738,A -85,B 0,C 180,E1 -31184.352,E2 -31184.352} C_VEL
LIN {X 0,Y 21.463,Z 376.288,A -85,B 0,C 180,E1 -31195.79,E2 -31195.79} C_VEL
LIN {X 0,Y 16.94,Z 378.525,A -85,B 0,C 180,E1 -31205.053,E2 -31205.053} C_VEL
LIN {X 0,Y 12.278,Z 380.421,A -85,B 0,C 180,E1 -31217.676,E2 -31217.676} C_VEL
LIN {X 0,Y 7.659,Z 383.495,A -85,B 0,C 180,E1 -31284.268,E2 -31284.268} C_VEL
LIN {X 0,Y 11.196,Z 384.735,A -85,B 0,C 180,E1 -31313.269,E2 -31313.269} C_VEL
LIN {X 0,Y 12.89,Z 385.053,A -85,B 0,C 180,E1 -31317.841,E2 -31317.841} C_VEL
LIN {X 0,Y 21.317,Z 386.375,A -85,B 0,C 180,E1 -31328.498,E2 -31328.498} C_VEL
LIN {X 0,Y 21.431,Z 386.415,A -85,B 0,C 180,E1 -31330.337,E2 -31330.337} C_VEL
LIN {X 0,Y 8.897,Z 384.438,A -85,B 0,C 180,E1 -31357.836,E2 -31357.836} C_VEL
LIN {X 0,Y 5.973,Z 382.86,A -85,B 0,C 180,E1 -31410.014,E2 -31410.014} C_VEL
LIN {X 0,Y 11.698,Z 379.499,A -85,B 0,C 180,E1 -31474.329,E2 -31474.329} C_VEL
LIN {X 0,Y 21.42,Z 375.011,A -85,B 0,C 180,E1 -31489.86,E2 -31489.86} C_VEL
LIN {X 0,Y 33.461,Z 368.18,A -85,B 0,C 180,E1 -31496.134,E2 -31496.134} C_VEL
LIN {X 0,Y 43.692,Z 360.879,A -85,B 0,C 180,E1 -31499.033,E2 -31499.033} C_VEL
LIN {X 0,Y 52.71,Z 353.087,A -85,B 0,C 180,E1 -31500.439,E2 -31500.439} C_VEL
LIN {X 0,Y 61.518,Z 343.833,A -85,B 0,C 180,E1 -31501.498,E2 -31501.498} C_VEL
LIN {X 0,Y 69.45,Z 333.574,A -85,B 0,C 180,E1 -31502.09,E2 -31502.09} C_VEL
LIN {X 0,Y 76.51,Z 322.168,A -85,B 0,C 180,E1 -31502.598,E2 -31502.598} C_VEL
LIN {X 0,Y 82.24,Z 310.424,A -85,B 0,C 180,E1 -31502.808,E2 -31502.808} C_VEL
LIN {X 0,Y 86.833,Z 297.617,A -85,B 0,C 180,E1 -31503.036,E2 -31503.036} C_VEL
LIN {X 0,Y 90.079,Z 284.266,A -85,B 0,C 180,E1 -31503.259,E2 -31503.259} C_VEL
LIN {X 0,Y 90.232,Z 283.261,A -85,B 0,C 180,E1 -31503.48,E2 -31503.48} C_VEL
LIN {X 0,Y 90.046,Z 280.362,A -85,B 0,C 180,E1 -31507.847,E2 -31507.847} C_VEL
LIN {X 0,Y 89.901,Z 280.389,A -85,B 0,C 180,E1 -31511.167,E2 -31511.167} C_VEL
LIN {X 0,Y 89.977,Z 281.56,A -85,B 0,C 180,E1 -31515.976,E2 -31515.976} C_VEL
LIN {X 0,Y 90.144,Z 283.274,A -85,B 0,C 180,E1 -31519.013,E2 -31519.013} C_VEL
LIN {X 0,Y 86.791,Z 297.138,A -85,B 0,C 180,E1 -31519.401,E2 -31519.401} C_VEL
LIN {X 0,Y 82.194,Z 309.937,A -85,B 0,C 180,E1 -31519.85,E2 -31519.85} C_VEL
LIN {X 0,Y 76.831,Z 321.07,A -85,B 0,C 180,E1 -31520.342,E2 -31520.342} C_VEL
LIN {X 0,Y 69.646,Z 332.77,A -85,B 0,C 180,E1 -31521.02,E2 -31521.02} C_VEL
LIN {X 0,Y 61.577,Z 343.283,A -85,B 0,C 180,E1 -31521.973,E2 -31521.973} C_VEL
LIN {X 0,Y 51.721,Z 353.545,A -85,B 0,C 180,E1 -31523.473,E2 -31523.473} C_VEL
LIN {X 0,Y 42.713,Z 361.194,A -85,B 0,C 180,E1 -31525.174,E2 -31525.174} C_VEL
LIN {X 0,Y 32.004,Z 368.669,A -85,B 0,C 180,E1 -31528.544,E2 -31528.544} C_VEL
LIN {X 0,Y 21.324,Z 374.614,A -85,B 0,C 180,E1 -31534.511,E2 -31534.511} C_VEL
LIN {X 0,Y 11.033,Z 379.295,A -85,B 0,C 180,E1 -31550.422,E2 -31550.422} C_VEL
LIN {X 0,Y 5.624,Z 382.842,A -85,B 0,C 180,E1 -31628.65,E2 -31628.65} C_VEL
LIN {X 0,Y 12.89,Z 385.053,A -85,B 0,C 180,E1 -31677.841,E2 -31677.841} C_VEL
LIN {X 0,Y 11.801,Z 384.968,A -85,B 0,C 180,E1 -31680.603,E2 -31680.603} C_VEL
LIN {X 0,Y 5.201,Z 383.643,A -85,B 0,C 180,E1 -31679.643,E2 -31679.643} C_VEL
LIN {X 0,Y 3.541,Z 381.263,A -85,B 0,C 180,E1 -31525.512,E2 -31525.512} C_VEL
LIN {X 0,Y 10.197,Z 378.945,A -85,B 0,C 180,E1 -31516.388,E2 -31516.388} C_VEL
LIN {X 0,Y 16.781,Z 376.219,A -85,B 0,C 180,E1 -31515.207,E2 -31515.207} C_VEL
LIN {X 0,Y 23.193,Z 373.097,A -85,B 0,C 180,E1 -31515.411,E2 -31515.411} C_VEL
LIN {X 0,Y 34.686,Z 366.372,A -85,B 0,C 180,E1 -31515.742,E2 -31515.742} C_VEL
LIN {X 0,Y 45.613,Z 358.273,A -85,B 0,C 180,E1 -31515.63,E2 -31515.63} C_VEL
LIN {X 0,Y 55.306,Z 349.346,A -85,B 0,C 180,E1 -31515.474,E2 -31515.474} C_VEL
LIN {X 0,Y 63.752,Z 339.821,A -85,B 0,C 180,E1 -31515.285,E2 -31515.285} C_VEL
LIN {X 0,Y 71,Z 329.821,A -85,B 0,C 180,E1 -31515.174,E2 -31515.174} C_VEL
LIN {X 0,Y 77.316,Z 318.969,A -85,B 0,C 180,E1 -31515.02,E2 -31515.02} C_VEL
LIN {X 0,Y 82.752,Z 306.975,A -85,B 0,C 180,E1 -31514.865,E2 -31514.865} C_VEL
LIN {X 0,Y 87.167,Z 293.725,A -85,B 0,C 180,E1 -31514.637,E2 -31514.637} C_VEL
LIN {X 0,Y 88.557,Z 288.094,A -85,B 0,C 180,E1 -31514.492,E2 -31514.492} C_VEL
LIN {X 0,Y 88.696,Z 287.188,A -85,B 0,C 180,E1 -31509.114,E2 -31509.114} C_VEL
LIN {X 0,Y 88.673,Z 287.776,A -85,B 0,C 180,E1 -31507.805,E2 -31507.805} C_VEL
LIN {X 0,Y 85.11,Z 300.721,A -85,B 0,C 180,E1 -31507.724,E2 -31507.724} C_VEL
LIN {X 0,Y 80.425,Z 312.712,A -85,B 0,C 180,E1 -31507.81,E2 -31507.81} C_VEL
LIN {X 0,Y 74.508,Z 324.277,A -85,B 0,C 180,E1 -31507.928,E2 -31507.928} C_VEL
LIN {X 0,Y 67.42,Z 335.195,A -85,B 0,C 180,E1 -31507.974,E2 -31507.974} C_VEL
LIN {X 0,Y 60.34,Z 344.079,A -85,B 0,C 180,E1 -31508.089,E2 -31508.089} C_VEL
LIN {X 0,Y 51.365,Z 353.339,A -85,B 0,C 180,E1 -31508.144,E2 -31508.144} C_VEL
LIN {X 0,Y 40.844,Z 362.149,A -85,B 0,C 180,E1 -31508.332,E2 -31508.332} C_VEL
LIN {X 0,Y 30.192,Z 369.302,A -85,B 0,C 180,E1 -31508.367,E2 -31508.367} C_VEL
LIN {X 0,Y 17.813,Z 375.765,A -85,B 0,C 180,E1 -31509.438,E2 -31509.438} C_VEL
